LIN {X 0,Y 367.15,Z 1229.112,A -85,B 0,C 180,E1 18985.265,E2 18985.265} C_VEL
LIN {X 0,Y 367.339,Z 1230.535,A -85,B 0,C 180,E1 18990,E2 18990} C_VEL
LIN {X 0,Y 367.173,Z 1229.12,A -85,B 0,C 180,E1 18994.734,E2 18994.734} C_VEL
LIN {X 0,Y 367.735,Z 1223.43,A -85,B 0,C 180,E1 19000.686,E2 19000.686} C_VEL
LIN {X 0,Y 369.708,Z 1212.061,A -85,B 0,C 180,E1 19007.286,E2 19007.286} C_VEL
LIN {X 0,Y 374.711,Z 1193.004,A -85,B 0,C 180,E1 19014.404,E2 19014.404} C_VEL
LIN {X 0,Y 382.386,Z 1169.034,A -85,B 0,C 180,E1 19020.677,E2 19020.677} C_VEL
LIN {X 0,Y 392.699,Z 1139.664,A -85,B 0,C 180,E1 19026.255,E2 19026.255} C_VEL
LIN {X 0,Y 404.453,Z 1104.956,A -85,B 0,C 180,E1 19031.092,E2 19031.092} C_VEL
LIN {X 0,Y 416.185,Z 1066.688,A -85,B 0,C 180,E1 19034.968,E2 19034.968} C_VEL
LIN {X 0,Y 426.949,Z 1024.996,A -85,B 0,C 180,E1 19037.984,E2 19037.984} C_VEL
LIN {X 0,Y 432.113,Z 1000.704,A -85,B 0,C 180,E1 19039.291,E2 19039.291} C_VEL
LIN {X 0,Y 431.695,Z 993.378,A -85,B 0,C 180,E1 19039.909,E2 19039.909} C_VEL
LIN {X 0,Y 427.323,Z 982.88,A -85,B 0,C 180,E1 19041.274,E2 19041.274} C_VEL
LIN {X 0,Y 415.984,Z 952.064,A -85,B 0,C 180,E1 19044.997,E2 19044.997} C_VEL
LIN {X 0,Y 400.09,Z 921.403,A -85,B 0,C 180,E1 19049.492,E2 19049.492} C_VEL
LIN {X 0,Y 385.069,Z 898.25,A -85,B 0,C 180,E1 19053.963,E2 19053.963} C_VEL
LIN {X 0,Y 372.467,Z 880.115,A -85,B 0,C 180,E1 19058.525,E2 19058.525} C_VEL
LIN {X 0,Y 367.434,Z 873.394,A -85,B 0,C 180,E1 19060.66,E2 19060.66} C_VEL
LIN {X 0,Y 363.503,Z 867.579,A -85,B 0,C 180,E1 19062.545,E2 19062.545} C_VEL
LIN {X 0,Y 358.526,Z 862.168,A -85,B 0,C 180,E1 19065.154,E2 19065.154} C_VEL
LIN {X 0,Y 358.075,Z 859.31,A -85,B 0,C 180,E1 19065.699,E2 19065.699} C_VEL
LIN {X 0,Y 358.617,Z 859.31,A -85,B 0,C 180,E1 19072.716,E2 19072.716} C_VEL
LIN {X 0,Y 359.258,Z 859.31,A -85,B 0,C 180,E1 19079.997,E2 19079.997} C_VEL
LIN {X 0,Y 358.638,Z 859.31,A -85,B 0,C 180,E1 19087.277,E2 19087.277} C_VEL
LIN {X 0,Y 358.029,Z 859.31,A -85,B 0,C 180,E1 19094.703,E2 19094.703} C_VEL
LIN {X 0,Y 357.661,Z 859.332,A -85,B 0,C 180,E1 19100.287,E2 19100.287} C_VEL
LIN {X 0,Y 359.157,Z 864.008,A -85,B 0,C 180,E1 19101.329,E2 19101.329} C_VEL
LIN {X 0,Y 363.357,Z 867.747,A -85,B 0,C 180,E1 19103.444,E2 19103.444} C_VEL
LIN {X 0,Y 366.991,Z 873.322,A -85,B 0,C 180,E1 19105.191,E2 19105.191} C_VEL
LIN {X 0,Y 369.225,Z 876.271,A -85,B 0,C 180,E1 19106.168,E2 19106.168} C_VEL
LIN {X 0,Y 379.086,Z 889.509,A -85,B 0,C 180,E1 19109.965,E2 19109.965} C_VEL
LIN {X 0,Y 395.189,Z 912.841,A -85,B 0,C 180,E1 19115,E2 19115} C_VEL
LIN {X 0,Y 413.421,Z 943.358,A -85,B 0,C 180,E1 19119.705,E2 19119.705} C_VEL
LIN {X 0,Y 427.964,Z 974.626,A -85,B 0,C 180,E1 19123.471,E2 19123.471} C_VEL
LIN {X 0,Y 431.637,Z 986.503,A -85,B 0,C 180,E1 19124.663,E2 19124.663} C_VEL
LIN {X 0,Y 424.084,Z 1024.913,A -85,B 0,C 180,E1 19126.278,E2 19126.278} C_VEL
LIN {X 0,Y 414.384,Z 1061.767,A -85,B 0,C 180,E1 19128.631,E2 19128.631} C_VEL
LIN {X 0,Y 403.385,Z 1095.493,A -85,B 0,C 180,E1 19131.699,E2 19131.699} C_VEL
LIN {X 0,Y 391.865,Z 1125.986,A -85,B 0,C 180,E1 19135.561,E2 19135.561} C_VEL
LIN {X 0,Y 380.389,Z 1153.684,A -85,B 0,C 180,E1 19140.465,E2 19140.465} C_VEL
LIN {X 0,Y 371.321,Z 1175.527,A -85,B 0,C 180,E1 19145.916,E2 19145.916} C_VEL
LIN {X 0,Y 364.796,Z 1192.186,A -85,B 0,C 180,E1 19151.849,E2 19151.849} C_VEL
LIN {X 0,Y 361.198,Z 1203.353,A -85,B 0,C 180,E1 19157.892,E2 19157.892} C_VEL
LIN {X 0,Y 359.855,Z 1208.915,A -85,B 0,C 180,E1 19162.743,E2 19162.743} C_VEL
LIN {X 0,Y 359.413,Z 1211.64,A -85,B 0,C 180,E1 19167.584,E2 19167.584} C_VEL
LIN {X 0,Y 359.465,Z 1211.596,A -85,B 0,C 180,E1 19172.416,E2 19172.416} C_VEL
LIN {X 0,Y 360.028,Z 1208.022,A -85,B 0,C 180,E1 19178.09,E2 19178.09} C_VEL
LIN {X 0,Y 362.386,Z 1199.251,A -85,B 0,C 180,E1 19184.53,E2 19184.53} C_VEL
LIN {X 0,Y 367.067,Z 1185.895,A -85,B 0,C 180,E1 19190.542,E2 19190.542} C_VEL
LIN {X 0,Y 374.831,Z 1166.721,A -85,B 0,C 180,E1 19196.404,E2 19196.404} C_VEL
LIN {X 0,Y 385.163,Z 1142.05,A -85,B 0,C 180,E1 19201.695,E2 19201.695} C_VEL
LIN {X 0,Y 396.787,Z 1113.062,A -85,B 0,C 180,E1 19206.125,E2 19206.125} C_VEL
LIN {X 0,Y 408.628,Z 1079.698,A -85,B 0,C 180,E1 19209.768,E2 19209.768} C_VEL
LIN {X 0,Y 419.448,Z 1043.217,A -85,B 0,C 180,E1 19212.567,E2 19212.567} C_VEL
LIN {X 0,Y 428.235,Z 1005.04,A -85,B 0,C 180,E1 19214.553,E2 19214.553} C_VEL
LIN {X 0,Y 431.34,Z 984.283,A -85,B 0,C 180,E1 19215.383,E2 19215.383} C_VEL
LIN {X 0,Y 417.794,Z 951.743,A -85,B 0,C 180,E1 19219.089,E2 19219.089} C_VEL
LIN {X 0,Y 400.846,Z 921.844,A -85,B 0,C 180,E1 19223.316,E2 19223.316} C_VEL
LIN {X 0,Y 385.133,Z 898.179,A -85,B 0,C 180,E1 19227.847,E2 19227.847} C_VEL
LIN {X 0,Y 375.352,Z 884.709,A -85,B 0,C 180,E1 19231.201,E2 19231.201} C_VEL
LIN {X 0,Y 371.503,Z 879.558,A -85,B 0,C 180,E1 19232.697,E2 19232.697} C_VEL
LIN {X 0,Y 367.256,Z 873.532,A -85,B 0,C 180,E1 19234.502,E2 19234.502} C_VEL
LIN {X 0,Y 363.334,Z 867.894,A -85,B 0,C 180,E1 19236.349,E2 19236.349} C_VEL
LIN {X 0,Y 357.895,Z 861.738,A -85,B 0,C 180,E1 19239.2,E2 19239.2} C_VEL
LIN {X 0,Y 357.537,Z 859.31,A -85,B 0,C 180,E1 19239.568,E2 19239.568} C_VEL
LIN {X 0,Y 358.034,Z 859.31,A -85,B 0,C 180,E1 19246.761,E2 19246.761} C_VEL
LIN {X 0,Y 358.648,Z 859.31,A -85,B 0,C 180,E1 19252.723,E2 19252.723} C_VEL
LIN {X 0,Y 359.263,Z 859.31,A -85,B 0,C 180,E1 19260.003,E2 19260.003} C_VEL
LIN {X 0,Y 358.62,Z 859.31,A -85,B 0,C 180,E1 19267.284,E2 19267.284} C_VEL
LIN {X 0,Y 358.065,Z 859.874,A -85,B 0,C 180,E1 19274.607,E2 19274.607} C_VEL
LIN {X 0,Y 360.037,Z 864.711,A -85,B 0,C 180,E1 19275.876,E2 19275.876} C_VEL
LIN {X 0,Y 363.614,Z 867.802,A -85,B 0,C 180,E1 19277.621,E2 19277.621} C_VEL
LIN {X 0,Y 367.718,Z 873.561,A -85,B 0,C 180,E1 19279.559,E2 19279.559} C_VEL
LIN {X 0,Y 378.979,Z 889.438,A -85,B 0,C 180,E1 19284.034,E2 19284.034} C_VEL
LIN {X 0,Y 394.773,Z 912.854,A -85,B 0,C 180,E1 19289.06,E2 19289.06} C_VEL
LIN {X 0,Y 410.649,Z 941.029,A -85,B 0,C 180,E1 19293.521,E2 19293.521} C_VEL
LIN {X 0,Y 423.673,Z 972.018,A -85,B 0,C 180,E1 19297.488,E2 19297.488} C_VEL
LIN {X 0,Y 428.621,Z 990.013,A -85,B 0,C 180,E1 19299.444,E2 19299.444} C_VEL
LIN {X 0,Y 419.597,Z 1031.759,A -85,B 0,C 180,E1 19301.677,E2 19301.677} C_VEL
LIN {X 0,Y 409.092,Z 1070.519,A -85,B 0,C 180,E1 19304.638,E2 19304.638} C_VEL
LIN {X 0,Y 397.997,Z 1105.491,A -85,B 0,C 180,E1 19308.274,E2 19308.274} C_VEL
LIN {X 0,Y 386.322,Z 1138.586,A -85,B 0,C 180,E1 19312.91,E2 19312.91} C_VEL
LIN {X 0,Y 375.347,Z 1168.687,A -85,B 0,C 180,E1 19318.683,E2 19318.683} C_VEL
LIN {X 0,Y 367.176,Z 1193.104,A -85,B 0,C 180,E1 19325.193,E2 19325.193} C_VEL
LIN {X 0,Y 361.975,Z 1211.802,A -85,B 0,C 180,E1 19332.332,E2 19332.332} C_VEL
LIN {X 0,Y 359.893,Z 1223.198,A -85,B 0,C 180,E1 19339.078,E2 19339.078} C_VEL
LIN {X 0,Y 359.249,Z 1228.908,A -85,B 0,C 180,E1 19345.161,E2 19345.161} C_VEL
LIN {X 0,Y 359.439,Z 1230.334,A -85,B 0,C 180,E1 19350,E2 19350} C_VEL
LIN {X 0,Y 359.271,Z 1228.917,A -85,B 0,C 180,E1 19354.839,E2 19354.839} C_VEL
LIN {X 0,Y 359.87,Z 1223.22,A -85,B 0,C 180,E1 19360.922,E2 19360.922} C_VEL
LIN {X 0,Y 362,Z 1211.84,A -85,B 0,C 180,E1 19367.666,E2 19367.666} C_VEL
LIN {X 0,Y 367.136,Z 1193.199,A -85,B 0,C 180,E1 19374.793,E2 19374.793} C_VEL
LIN {X 0,Y 375.333,Z 1168.767,A -85,B 0,C 180,E1 19381.318,E2 19381.318} C_VEL
LIN {X 0,Y 386.374,Z 1138.707,A -85,B 0,C 180,E1 19387.083,E2 19387.083} C_VEL
LIN {X 0,Y 398.576,Z 1103.925,A -85,B 0,C 180,E1 19391.942,E2 19391.942} C_VEL
LIN {X 0,Y 410.79,Z 1065.255,A -85,B 0,C 180,E1 19395.85,E2 19395.85} C_VEL
LIN {X 0,Y 422.083,Z 1022.173,A -85,B 0,C 180,E1 19398.93,E2 19398.93} C_VEL
LIN {X 0,Y 428.825,Z 988.285,A -85,B 0,C 180,E1 19400.675,E2 19400.675} C_VEL
LIN {X 0,Y 427.323,Z 982.88,A -85,B 0,C 180,E1 19401.274,E2 19401.274} C_VEL
LIN {X 0,Y 422.821,Z 974.863,A -85,B 0,C 180,E1 19402.536,E2 19402.536} C_VEL
LIN {X 0,Y 414.499,Z 964.488,A -85,B 0,C 180,E1 19404.576,E2 19404.576} C_VEL
LIN {X 0,Y 413.821,Z 962.982,A -85,B 0,C 180,E1 19404.78,E2 19404.78} C_VEL
LIN {X 0,Y 399.432,Z 932.446,A -85,B 0,C 180,E1 19409.199,E2 19409.199} C_VEL
LIN {X 0,Y 383.451,Z 906.31,A -85,B 0,C 180,E1 19414.081,E2 19414.081} C_VEL
LIN {X 0,Y 369.915,Z 886.915,A -85,B 0,C 180,E1 19419.077,E2 19419.077} C_VEL
LIN {X 0,Y 364.832,Z 880.19,A -85,B 0,C 180,E1 19421.303,E2 19421.303} C_VEL
LIN {X 0,Y 360.151,Z 873.645,A -85,B 0,C 180,E1 19423.659,E2 19423.659} C_VEL
LIN {X 0,Y 356.32,Z 868.398,A -85,B 0,C 180,E1 19425.853,E2 19425.853} C_VEL
LIN {X 0,Y 355.113,Z 866.619,A -85,B 0,C 180,E1 19426.621,E2 19426.621} C_VEL
LIN {X 0,Y 350.857,Z 862.095,A -85,B 0,C 180,E1 19429.58,E2 19429.58} C_VEL
LIN {X 0,Y 350.463,Z 859.31,A -85,B 0,C 180,E1 19430.354,E2 19430.354} C_VEL
LIN {X 0,Y 351.103,Z 859.31,A -85,B 0,C 180,E1 19437.524,E2 19437.524} C_VEL
LIN {X 0,Y 351.143,Z 859.31,A -85,B 0,C 180,E1 19442.469,E2 19442.469} C_VEL
LIN {X 0,Y 350.438,Z 859.31,A -85,B 0,C 180,E1 19449.954,E2 19449.954} C_VEL
LIN {X 0,Y 350.018,Z 859.869,A -85,B 0,C 180,E1 19455.691,E2 19455.691} C_VEL
LIN {X 0,Y 352.008,Z 864.599,A -85,B 0,C 180,E1 19457.444,E2 19457.444} C_VEL
LIN {X 0,Y 355.863,Z 867.923,A -85,B 0,C 180,E1 19459.907,E2 19459.907} C_VEL
LIN {X 0,Y 359.622,Z 873.5,A -85,B 0,C 180,E1 19462.115,E2 19462.115} C_VEL
LIN {X 0,Y 361.689,Z 875.929,A -85,B 0,C 180,E1 19463.174,E2 19463.174} C_VEL
LIN {X 0,Y 367.943,Z 884.815,A -85,B 0,C 180,E1 19466.102,E2 19466.102} C_VEL
LIN {X 0,Y 377.036,Z 897.067,A -85,B 0,C 180,E1 19469.647,E2 19469.647} C_VEL
LIN {X 0,Y 392.135,Z 919.205,A -85,B 0,C 180,E1 19474.485,E2 19474.485} C_VEL
LIN {X 0,Y 409.719,Z 949.301,A -85,B 0,C 180,E1 19479.203,E2 19479.203} C_VEL
LIN {X 0,Y 423.434,Z 980.427,A -85,B 0,C 180,E1 19483.058,E2 19483.058} C_VEL
LIN {X 0,Y 425.993,Z 988.977,A -85,B 0,C 180,E1 19483.955,E2 19483.955} C_VEL
LIN {X 0,Y 418.022,Z 1027.436,A -85,B 0,C 180,E1 19485.628,E2 19485.628} C_VEL
LIN {X 0,Y 407.954,Z 1064.073,A -85,B 0,C 180,E1 19488.042,E2 19488.042} C_VEL
LIN {X 0,Y 396.34,Z 1098.126,A -85,B 0,C 180,E1 19491.241,E2 19491.241} C_VEL
LIN {X 0,Y 384.591,Z 1128,A -85,B 0,C 180,E1 19495.159,E2 19495.159} C_VEL
LIN {X 0,Y 373.441,Z 1153.942,A -85,B 0,C 180,E1 19499.859,E2 19499.859} C_VEL
LIN {X 0,Y 364.005,Z 1175.757,A -85,B 0,C 180,E1 19505.4,E2 19505.4} C_VEL
LIN {X 0,Y 357.194,Z 1192.404,A -85,B 0,C 180,E1 19511.448,E2 19511.448} C_VEL
LIN {X 0,Y 353.418,Z 1203.561,A -85,B 0,C 180,E1 19517.621,E2 19517.621} C_VEL
LIN {X 0,Y 351.979,Z 1209.12,A -85,B 0,C 180,E1 19522.58,E2 19522.58} C_VEL
LIN {X 0,Y 351.514,Z 1211.843,A -85,B 0,C 180,E1 19527.53,E2 19527.53} C_VEL
LIN {X 0,Y 351.564,Z 1211.798,A -85,B 0,C 180,E1 19532.471,E2 19532.471} C_VEL
LIN {X 0,Y 352.232,Z 1208.057,A -85,B 0,C 180,E1 19538.455,E2 19538.455} C_VEL
LIN {X 0,Y 354.68,Z 1199.462,A -85,B 0,C 180,E1 19544.853,E2 19544.853} C_VEL
LIN {X 0,Y 359.6,Z 1186.123,A -85,B 0,C 180,E1 19550.988,E2 19550.988} C_VEL
LIN {X 0,Y 367.684,Z 1166.975,A -85,B 0,C 180,E1 19556.958,E2 19556.958} C_VEL
LIN {X 0,Y 378.689,Z 1141.618,A -85,B 0,C 180,E1 19562.46,E2 19562.46} C_VEL
LIN {X 0,Y 390.707,Z 1112.592,A -85,B 0,C 180,E1 19566.918,E2 19566.918} C_VEL
LIN {X 0,Y 402.592,Z 1080.169,A -85,B 0,C 180,E1 19570.486,E2 19570.486} C_VEL
LIN {X 0,Y 413.994,Z 1042.731,A -85,B 0,C 180,E1 19573.375,E2 19573.375} C_VEL
LIN {X 0,Y 423.128,Z 1003.727,A -85,B 0,C 180,E1 19575.393,E2 19575.393} C_VEL
LIN {X 0,Y 425.615,Z 987.109,A -85,B 0,C 180,E1 19576.086,E2 19576.086} C_VEL
LIN {X 0,Y 412.44,Z 954.819,A -85,B 0,C 180,E1 19579.919,E2 19579.919} C_VEL
LIN {X 0,Y 396.061,Z 925.668,A -85,B 0,C 180,E1 19584.252,E2 19584.252} C_VEL
LIN {X 0,Y 379.708,Z 900.578,A -85,B 0,C 180,E1 19589.262,E2 19589.262} C_VEL
LIN {X 0,Y 368.895,Z 886.075,A -85,B 0,C 180,E1 19593.314,E2 19593.314} C_VEL
LIN {X 0,Y 364.408,Z 880.099,A -85,B 0,C 180,E1 19595.276,E2 19595.276} C_VEL
LIN {X 0,Y 360.295,Z 873.963,A -85,B 0,C 180,E1 19597.34,E2 19597.34} C_VEL
LIN {X 0,Y 355.922,Z 868.494,A -85,B 0,C 180,E1 19599.772,E2 19599.772} C_VEL
LIN {X 0,Y 354.505,Z 866.563,A -85,B 0,C 180,E1 19600.663,E2 19600.663} C_VEL
LIN {X 0,Y 350.327,Z 861.978,A -85,B 0,C 180,E1 19603.599,E2 19603.599} C_VEL
LIN {X 0,Y 349.914,Z 859.31,A -85,B 0,C 180,E1 19604.305,E2 19604.305} C_VEL
LIN {X 0,Y 350.437,Z 859.31,A -85,B 0,C 180,E1 19610.046,E2 19610.046} C_VEL
LIN {X 0,Y 351.109,Z 859.31,A -85,B 0,C 180,E1 19617.531,E2 19617.531} C_VEL
LIN {X 0,Y 351.148,Z 859.31,A -85,B 0,C 180,E1 19622.476,E2 19622.476} C_VEL
LIN {X 0,Y 350.42,Z 859.698,A -85,B 0,C 180,E1 19630.118,E2 19630.118} C_VEL
LIN {X 0,Y 352.122,Z 864.387,A -85,B 0,C 180,E1 19631.638,E2 19631.638} C_VEL
LIN {X 0,Y 356.14,Z 867.806,A -85,B 0,C 180,E1 19634.158,E2 19634.158} C_VEL
LIN {X 0,Y 359.617,Z 873.291,A -85,B 0,C 180,E1 19636.209,E2 19636.209} C_VEL
LIN {X 0,Y 361.893,Z 875.863,A -85,B 0,C 180,E1 19637.356,E2 19637.356} C_VEL
LIN {X 0,Y 367.733,Z 884.15,A -85,B 0,C 180,E1 19640.107,E2 19640.107} C_VEL
LIN {X 0,Y 376.638,Z 896.626,A -85,B 0,C 180,E1 19643.641,E2 19643.641} C_VEL
LIN {X 0,Y 391.562,Z 919.088,A -85,B 0,C 180,E1 19648.53,E2 19648.53} C_VEL
LIN {X 0,Y 406.621,Z 946.779,A -85,B 0,C 180,E1 19653.019,E2 19653.019} C_VEL
LIN {X 0,Y 418.988,Z 977.742,A -85,B 0,C 180,E1 19657.083,E2 19657.083} C_VEL
LIN {X 0,Y 422.934,Z 992.326,A -85,B 0,C 180,E1 19658.745,E2 19658.745} C_VEL
LIN {X 0,Y 412.869,Z 1036.702,A -85,B 0,C 180,E1 19661.203,E2 19661.203} C_VEL
LIN {X 0,Y 400.633,Z 1079.007,A -85,B 0,C 180,E1 19664.64,E2 19664.64} C_VEL
LIN {X 0,Y 387.942,Z 1116.268,A -85,B 0,C 180,E1 19668.892,E2 19668.892} C_VEL
LIN {X 0,Y 375.255,Z 1150.031,A -85,B 0,C 180,E1 19674.225,E2 19674.225} C_VEL
LIN {X 0,Y 365.282,Z 1177.147,A -85,B 0,C 180,E1 19680.145,E2 19680.145} C_VEL
LIN {X 0,Y 357.663,Z 1199.514,A -85,B 0,C 180,E1 19686.927,E2 19686.927} C_VEL
LIN {X 0,Y 353.375,Z 1215.207,A -85,B 0,C 180,E1 19693.816,E2 19693.816} C_VEL
LIN {X 0,Y 351.812,Z 1224.499,A -85,B 0,C 180,E1 19700.079,E2 19700.079} C_VEL
LIN {X 0,Y 351.35,Z 1228.705,A -85,B 0,C 180,E1 19705.051,E2 19705.051} C_VEL
LIN {X 0,Y 351.54,Z 1230.132,A -85,B 0,C 180,E1 19710,E2 19710} C_VEL
LIN {X 0,Y 351.37,Z 1228.714,A -85,B 0,C 180,E1 19714.948,E2 19714.948} C_VEL
LIN {X 0,Y 352.005,Z 1223.01,A -85,B 0,C 180,E1 19721.169,E2 19721.169} C_VEL
LIN {X 0,Y 354.296,Z 1211.619,A -85,B 0,C 180,E1 19728.064,E2 19728.064} C_VEL
LIN {X 0,Y 359.767,Z 1192.96,A -85,B 0,C 180,E1 19735.337,E2 19735.337} C_VEL
LIN {X 0,Y 368.369,Z 1168.5,A -85,B 0,C 180,E1 19741.979,E2 19741.979} C_VEL
LIN {X 0,Y 379.889,Z 1138.391,A -85,B 0,C 180,E1 19747.826,E2 19747.826} C_VEL
LIN {X 0,Y 392.422,Z 1103.855,A -85,B 0,C 180,E1 19752.701,E2 19752.701} C_VEL
LIN {X 0,Y 405.166,Z 1064.689,A -85,B 0,C 180,E1 19756.68,E2 19756.68} C_VEL
LIN {X 0,Y 416.483,Z 1022.91,A -85,B 0,C 180,E1 19759.679,E2 19759.679} C_VEL
LIN {X 0,Y 423.112,Z 991.352,A -85,B 0,C 180,E1 19761.329,E2 19761.329} C_VEL
LIN {X 0,Y 413.821,Z 962.982,A -85,B 0,C 180,E1 19764.78,E2 19764.78} C_VEL
LIN {X 0,Y 408.724,Z 955.768,A -85,B 0,C 180,E1 19766.131,E2 19766.131} C_VEL
LIN {X 0,Y 399.285,Z 945.576,A -85,B 0,C 180,E1 19768.576,E2 19768.576} C_VEL
LIN {X 0,Y 384.747,Z 919.229,A -85,B 0,C 180,E1 19773.231,E2 19773.231} C_VEL
LIN {X 0,Y 368.413,Z 894.706,A -85,B 0,C 180,E1 19779.224,E2 19779.224} C_VEL
LIN {X 0,Y 358.317,Z 881.083,A -85,B 0,C 180,E1 19784.046,E2 19784.046} C_VEL
LIN {X 0,Y 354.379,Z 875.295,A -85,B 0,C 180,E1 19786.398,E2 19786.398} C_VEL
LIN {X 0,Y 349.218,Z 869.207,A -85,B 0,C 180,E1 19790.083,E2 19790.083} C_VEL
LIN {X 0,Y 348.367,Z 866.925,A -85,B 0,C 180,E1 19790.927,E2 19790.927} C_VEL
LIN {X 0,Y 343.482,Z 861.831,A -85,B 0,C 180,E1 19796.52,E2 19796.52} C_VEL
LIN {X 0,Y 343.23,Z 859.31,A -85,B 0,C 180,E1 19797.783,E2 19797.783} C_VEL
LIN {X 0,Y 343.227,Z 859.31,A -85,B 0,C 180,E1 19802.526,E2 19802.526} C_VEL
LIN {X 0,Y 342.745,Z 859.975,A -85,B 0,C 180,E1 19807.856,E2 19807.856} C_VEL
LIN {X 0,Y 345.119,Z 865.303,A -85,B 0,C 180,E1 19812.031,E2 19812.031} C_VEL
LIN {X 0,Y 348.552,Z 867.994,A -85,B 0,C 180,E1 19815.346,E2 19815.346} C_VEL
LIN {X 0,Y 352.066,Z 873.596,A -85,B 0,C 180,E1 19818.174,E2 19818.174} C_VEL
LIN {X 0,Y 354.361,Z 875.948,A -85,B 0,C 180,E1 19819.639,E2 19819.639} C_VEL
LIN {X 0,Y 359.026,Z 881.65,A -85,B 0,C 180,E1 19822.315,E2 19822.315} C_VEL
LIN {X 0,Y 373.94,Z 902.767,A -85,B 0,C 180,E1 19828.918,E2 19828.918} C_VEL
LIN {X 0,Y 389.418,Z 926.115,A -85,B 0,C 180,E1 19834.056,E2 19834.056} C_VEL
LIN {X 0,Y 405.851,Z 955.267,A -85,B 0,C 180,E1 19838.721,E2 19838.721} C_VEL
LIN {X 0,Y 418.768,Z 986.191,A -85,B 0,C 180,E1 19842.651,E2 19842.651} C_VEL
LIN {X 0,Y 420.308,Z 992.169,A -85,B 0,C 180,E1 19843.256,E2 19843.256} C_VEL
LIN {X 0,Y 411.574,Z 1031.755,A -85,B 0,C 180,E1 19845.055,E2 19845.055} C_VEL
LIN {X 0,Y 400.039,Z 1070.982,A -85,B 0,C 180,E1 19847.802,E2 19847.802} C_VEL
LIN {X 0,Y 387.602,Z 1105.211,A -85,B 0,C 180,E1 19851.281,E2 19851.281} C_VEL
LIN {X 0,Y 374.579,Z 1136.428,A -85,B 0,C 180,E1 19855.8,E2 19855.8} C_VEL
LIN {X 0,Y 362.821,Z 1162.416,A -85,B 0,C 180,E1 19861.134,E2 19861.134} C_VEL
LIN {X 0,Y 354.356,Z 1181.426,A -85,B 0,C 180,E1 19866.629,E2 19866.629} C_VEL
LIN {X 0,Y 347.87,Z 1197.306,A -85,B 0,C 180,E1 19873.333,E2 19873.333} C_VEL
LIN {X 0,Y 344.701,Z 1206.912,A -85,B 0,C 180,E1 19879.873,E2 19879.873} C_VEL
LIN {X 0,Y 343.776,Z 1211.03,A -85,B 0,C 180,E1 19884.943,E2 19884.943} C_VEL
LIN {X 0,Y 343.666,Z 1212.365,A -85,B 0,C 180,E1 19890,E2 19890} C_VEL
LIN {X 0,Y 343.792,Z 1210.956,A -85,B 0,C 180,E1 19895.058,E2 19895.058} C_VEL
LIN {X 0,Y 345.209,Z 1205.29,A -85,B 0,C 180,E1 19901.393,E2 19901.393} C_VEL
LIN {X 0,Y 349.176,Z 1193.679,A -85,B 0,C 180,E1 19908.338,E2 19908.338} C_VEL
LIN {X 0,Y 356.801,Z 1175.663,A -85,B 0,C 180,E1 19915.131,E2 19915.131} C_VEL
LIN {X 0,Y 367.379,Z 1152.445,A -85,B 0,C 180,E1 19921.036,E2 19921.036} C_VEL
LIN {X 0,Y 379.761,Z 1124.211,A -85,B 0,C 180,E1 19926.054,E2 19926.054} C_VEL
LIN {X 0,Y 392.566,Z 1091.951,A -85,B 0,C 180,E1 19930.101,E2 19930.101} C_VEL
LIN {X 0,Y 404.763,Z 1055.846,A -85,B 0,C 180,E1 19933.27,E2 19933.27} C_VEL
LIN {X 0,Y 414.816,Z 1018.042,A -85,B 0,C 180,E1 19935.553,E2 19935.553} C_VEL
LIN {X 0,Y 419.92,Z 989.876,A -85,B 0,C 180,E1 19936.816,E2 19936.816} C_VEL
LIN {X 0,Y 407.158,Z 958.008,A -85,B 0,C 180,E1 19940.768,E2 19940.768} C_VEL
LIN {X 0,Y 391.258,Z 929.144,A -85,B 0,C 180,E1 19945.251,E2 19945.251} C_VEL
LIN {X 0,Y 375.727,Z 905.574,A -85,B 0,C 180,E1 19950.24,E2 19950.24} C_VEL
LIN {X 0,Y 363.526,Z 888.276,A -85,B 0,C 180,E1 19955.212,E2 19955.212} C_VEL
LIN {X 0,Y 357.749,Z 880.867,A -85,B 0,C 180,E1 19958.108,E2 19958.108} C_VEL
LIN {X 0,Y 352.815,Z 874.13,A -85,B 0,C 180,E1 19961.088,E2 19961.088} C_VEL
LIN {X 0,Y 348.623,Z 868.766,A -85,B 0,C 180,E1 19964.206,E2 19964.206} C_VEL
LIN {X 0,Y 347.596,Z 866.844,A -85,B 0,C 180,E1 19965.156,E2 19965.156} C_VEL
LIN {X 0,Y 342.899,Z 861.607,A -85,B 0,C 180,E1 19970.708,E2 19970.708} C_VEL
LIN {X 0,Y 342.649,Z 859.31,A -85,B 0,C 180,E1 19971.742,E2 19971.742} C_VEL
LIN {X 0,Y 343.194,Z 859.31,A -85,B 0,C 180,E1 19977.474,E2 19977.474} C_VEL
LIN {X 0,Y 343.175,Z 860.095,A -85,B 0,C 180,E1 19983.246,E2 19983.246} C_VEL
LIN {X 0,Y 345.821,Z 865.525,A -85,B 0,C 180,E1 19987.04,E2 19987.04} C_VEL
LIN {X 0,Y 348.86,Z 868.02,A -85,B 0,C 180,E1 19989.769,E2 19989.769} C_VEL
LIN {X 0,Y 352.254,Z 873.421,A -85,B 0,C 180,E1 19992.421,E2 19992.421} C_VEL
LIN {X 0,Y 354.487,Z 875.664,A -85,B 0,C 180,E1 19993.834,E2 19993.834} C_VEL
LIN {X 0,Y 358.94,Z 881.458,A -85,B 0,C 180,E1 19996.398,E2 19996.398} C_VEL
LIN {X 0,Y 369.672,Z 896.846,A -85,B 0,C 180,E1 20001.409,E2 20001.409} C_VEL
LIN {X 0,Y 384.948,Z 919.742,A -85,B 0,C 180,E1 20006.912,E2 20006.912} C_VEL
LIN {X 0,Y 399.196,Z 945.574,A -85,B 0,C 180,E1 20011.456,E2 20011.456} C_VEL
LIN {X 0,Y 411.296,Z 974.691,A -85,B 0,C 180,E1 20015.577,E2 20015.577} C_VEL
LIN {X 0,Y 417.119,Z 995.397,A -85,B 0,C 180,E1 20018.069,E2 20018.069} C_VEL
LIN {X 0,Y 406.939,Z 1038.429,A -85,B 0,C 180,E1 20020.509,E2 20020.509} C_VEL
LIN {X 0,Y 394.695,Z 1079.379,A -85,B 0,C 180,E1 20023.886,E2 20023.886} C_VEL
LIN {X 0,Y 382.128,Z 1115.152,A -85,B 0,C 180,E1 20027.99,E2 20027.99} C_VEL
LIN {X 0,Y 369.263,Z 1148.207,A -85,B 0,C 180,E1 20033.195,E2 20033.195} C_VEL
LIN {X 0,Y 358.197,Z 1176.882,A -85,B 0,C 180,E1 20039.493,E2 20039.493} C_VEL
LIN {X 0,Y 350.13,Z 1199.472,A -85,B 0,C 180,E1 20046.476,E2 20046.476} C_VEL
LIN {X 0,Y 345.378,Z 1216.191,A -85,B 0,C 180,E1 20054.085,E2 20054.085} C_VEL
LIN {X 0,Y 343.798,Z 1225.573,A -85,B 0,C 180,E1 20061.126,E2 20061.126} C_VEL
LIN {X 0,Y 343.566,Z 1229.569,A -85,B 0,C 180,E1 20067.472,E2 20067.472} C_VEL
LIN {X 0,Y 343.558,Z 1229.571,A -85,B 0,C 180,E1 20072.528,E2 20072.528} C_VEL
LIN {X 0,Y 343.784,Z 1225.593,A -85,B 0,C 180,E1 20078.874,E2 20078.874} C_VEL
LIN {X 0,Y 345.428,Z 1216.227,A -85,B 0,C 180,E1 20085.912,E2 20085.912} C_VEL
LIN {X 0,Y 350.103,Z 1199.529,A -85,B 0,C 180,E1 20093.525,E2 20093.525} C_VEL
LIN {X 0,Y 358.191,Z 1176.962,A -85,B 0,C 180,E1 20100.507,E2 20100.507} C_VEL
LIN {X 0,Y 369.279,Z 1148.306,A -85,B 0,C 180,E1 20106.808,E2 20106.808} C_VEL
LIN {X 0,Y 382.144,Z 1115.276,A -85,B 0,C 180,E1 20112.015,E2 20112.015} C_VEL
LIN {X 0,Y 395.398,Z 1077.37,A -85,B 0,C 180,E1 20116.333,E2 20116.333} C_VEL
LIN {X 0,Y 407.775,Z 1035.881,A -85,B 0,C 180,E1 20119.67,E2 20119.67} C_VEL
LIN {X 0,Y 417.351,Z 994.067,A -85,B 0,C 180,E1 20122.039,E2 20122.039} C_VEL
LIN {X 0,Y 407.347,Z 963.466,A -85,B 0,C 180,E1 20125.936,E2 20125.936} C_VEL
LIN {X 0,Y 399.285,Z 945.576,A -85,B 0,C 180,E1 20128.576,E2 20128.576} C_VEL
LIN {X 0,Y 395.886,Z 941.099,A -85,B 0,C 180,E1 20129.545,E2 20129.545} C_VEL
LIN {X 0,Y 385.453,Z 931.977,A -85,B 0,C 180,E1 20132.478,E2 20132.478} C_VEL
LIN {X 0,Y 384.704,Z 930.725,A -85,B 0,C 180,E1 20132.724,E2 20132.724} C_VEL
LIN {X 0,Y 369.828,Z 907.382,A -85,B 0,C 180,E1 20138.127,E2 20138.127} C_VEL
LIN {X 0,Y 360.709,Z 894.477,A -85,B 0,C 180,E1 20142.191,E2 20142.191} C_VEL
LIN {X 0,Y 356.09,Z 888.129,A -85,B 0,C 180,E1 20144.656,E2 20144.656} C_VEL
LIN {X 0,Y 351.522,Z 881.565,A -85,B 0,C 180,E1 20147.553,E2 20147.553} C_VEL
LIN {X 0,Y 347.536,Z 876.057,A -85,B 0,C 180,E1 20150.668,E2 20150.668} C_VEL
LIN {X 0,Y 346.293,Z 874.345,A -85,B 0,C 180,E1 20151.823,E2 20151.823} C_VEL
LIN {X 0,Y 342.162,Z 868.741,A -85,B 0,C 180,E1 20157.221,E2 20157.221} C_VEL
LIN {X 0,Y 341.876,Z 867.092,A -85,B 0,C 180,E1 20158.092,E2 20158.092} C_VEL
LIN {X 0,Y 341.658,Z 867.792,A -85,B 0,C 180,E1 20167.564,E2 20167.564} C_VEL
LIN {X 0,Y 344.745,Z 873.663,A -85,B 0,C 180,E1 20172.689,E2 20172.689} C_VEL
LIN {X 0,Y 347.157,Z 875.681,A -85,B 0,C 180,E1 20175.003,E2 20175.003} C_VEL
LIN {X 0,Y 351.299,Z 881.641,A -85,B 0,C 180,E1 20178.311,E2 20178.311} C_VEL
LIN {X 0,Y 353.443,Z 884.854,A -85,B 0,C 180,E1 20179.743,E2 20179.743} C_VEL
LIN {X 0,Y 358.422,Z 891.44,A -85,B 0,C 180,E1 20182.6,E2 20182.6} C_VEL
LIN {X 0,Y 368.259,Z 905.192,A -85,B 0,C 180,E1 20187.149,E2 20187.149} C_VEL
LIN {X 0,Y 382.456,Z 926.004,A -85,B 0,C 180,E1 20192.274,E2 20192.274} C_VEL
LIN {X 0,Y 398.995,Z 955.04,A -85,B 0,C 180,E1 20197.327,E2 20197.327} C_VEL
LIN {X 0,Y 412.058,Z 985.78,A -85,B 0,C 180,E1 20201.5,E2 20201.5} C_VEL
LIN {X 0,Y 414.496,Z 995.633,A -85,B 0,C 180,E1 20202.559,E2 20202.559} C_VEL
LIN {X 0,Y 405.381,Z 1034.858,A -85,B 0,C 180,E1 20204.415,E2 20204.415} C_VEL
LIN {X 0,Y 394.096,Z 1071.77,A -85,B 0,C 180,E1 20207.06,E2 20207.06} C_VEL
LIN {X 0,Y 381.468,Z 1105.557,A -85,B 0,C 180,E1 20210.539,E2 20210.539} C_VEL
LIN {X 0,Y 368.628,Z 1135.395,A -85,B 0,C 180,E1 20214.867,E2 20214.867} C_VEL
LIN {X 0,Y 356.583,Z 1161.119,A -85,B 0,C 180,E1 20220.118,E2 20220.118} C_VEL
LIN {X 0,Y 346.843,Z 1182.013,A -85,B 0,C 180,E1 20226.234,E2 20226.234} C_VEL
LIN {X 0,Y 340.222,Z 1197.517,A -85,B 0,C 180,E1 20232.947,E2 20232.947} C_VEL
LIN {X 0,Y 336.879,Z 1207.118,A -85,B 0,C 180,E1 20239.635,E2 20239.635} C_VEL
LIN {X 0,Y 335.882,Z 1211.234,A -85,B 0,C 180,E1 20244.824,E2 20244.824} C_VEL
LIN {X 0,Y 335.767,Z 1212.567,A -85,B 0,C 180,E1 20250,E2 20250} C_VEL
LIN {X 0,Y 335.9,Z 1211.16,A -85,B 0,C 180,E1 20255.177,E2 20255.177} C_VEL
LIN {X 0,Y 337.405,Z 1205.496,A -85,B 0,C 180,E1 20261.66,E2 20261.66} C_VEL
LIN {X 0,Y 341.583,Z 1193.896,A -85,B 0,C 180,E1 20268.761,E2 20268.761} C_VEL
LIN {X 0,Y 349.556,Z 1175.893,A -85,B 0,C 180,E1 20275.69,E2 20275.69} C_VEL
LIN {X 0,Y 360.526,Z 1152.712,A -85,B 0,C 180,E1 20281.694,E2 20281.694} C_VEL
LIN {X 0,Y 373.346,Z 1124.544,A -85,B 0,C 180,E1 20286.774,E2 20286.774} C_VEL
LIN {X 0,Y 386.536,Z 1092.376,A -85,B 0,C 180,E1 20290.858,E2 20290.858} C_VEL
LIN {X 0,Y 398.952,Z 1056.855,A -85,B 0,C 180,E1 20294.013,E2 20294.013} C_VEL
LIN {X 0,Y 409.453,Z 1018.495,A -85,B 0,C 180,E1 20296.359,E2 20296.359} C_VEL
LIN {X 0,Y 414.42,Z 993.295,A -85,B 0,C 180,E1 20297.492,E2 20297.492} C_VEL
LIN {X 0,Y 402.582,Z 962.63,A -85,B 0,C 180,E1 20301.451,E2 20301.451} C_VEL
LIN {X 0,Y 387.595,Z 934.527,A -85,B 0,C 180,E1 20305.953,E2 20305.953} C_VEL
LIN {X 0,Y 372.426,Z 911.105,A -85,B 0,C 180,E1 20311.037,E2 20311.037} C_VEL
LIN {X 0,Y 360.913,Z 894.93,A -85,B 0,C 180,E1 20315.929,E2 20315.929} C_VEL
LIN {X 0,Y 355.904,Z 888.152,A -85,B 0,C 180,E1 20318.547,E2 20318.547} C_VEL
LIN {X 0,Y 351.234,Z 881.677,A -85,B 0,C 180,E1 20321.465,E2 20321.465} C_VEL
LIN {X 0,Y 347.03,Z 875.776,A -85,B 0,C 180,E1 20324.743,E2 20324.743} C_VEL
LIN {X 0,Y 341.598,Z 868.426,A -85,B 0,C 180,E1 20331.476,E2 20331.476} C_VEL
LIN {X 0,Y 341.277,Z 867.066,A -85,B 0,C 180,E1 20332.437,E2 20332.437} C_VEL
LIN {X 0,Y 341.947,Z 867.494,A -85,B 0,C 180,E1 20342.781,E2 20342.781} C_VEL
LIN {X 0,Y 344.73,Z 873.331,A -85,B 0,C 180,E1 20346.944,E2 20346.944} C_VEL
LIN {X 0,Y 347.398,Z 875.658,A -85,B 0,C 180,E1 20349.415,E2 20349.415} C_VEL
LIN {X 0,Y 351.274,Z 881.398,A -85,B 0,C 180,E1 20352.456,E2 20352.456} C_VEL
LIN {X 0,Y 353.287,Z 884.306,A -85,B 0,C 180,E1 20353.803,E2 20353.803} C_VEL
LIN {X 0,Y 358.673,Z 891.598,A -85,B 0,C 180,E1 20356.884,E2 20356.884} C_VEL
LIN {X 0,Y 367.62,Z 904.242,A -85,B 0,C 180,E1 20361.06,E2 20361.06} C_VEL
LIN {X 0,Y 381.953,Z 926.32,A -85,B 0,C 180,E1 20366.424,E2 20366.424} C_VEL
LIN {X 0,Y 395.623,Z 952.156,A -85,B 0,C 180,E1 20371.065,E2 20371.065} C_VEL
LIN {X 0,Y 406.919,Z 981.13,A -85,B 0,C 180,E1 20375.245,E2 20375.245} C_VEL
LIN {X 0,Y 411.345,Z 998.216,A -85,B 0,C 180,E1 20377.362,E2 20377.362} C_VEL
LIN {X 0,Y 401.36,Z 1039.063,A -85,B 0,C 180,E1 20379.719,E2 20379.719} C_VEL
LIN {X 0,Y 388.82,Z 1079.685,A -85,B 0,C 180,E1 20383.098,E2 20383.098} C_VEL
LIN {X 0,Y 375.298,Z 1116.87,A -85,B 0,C 180,E1 20387.445,E2 20387.445} C_VEL
LIN {X 0,Y 361.93,Z 1149.843,A -85,B 0,C 180,E1 20392.789,E2 20392.789} C_VEL
LIN {X 0,Y 351.16,Z 1176.617,A -85,B 0,C 180,E1 20398.814,E2 20398.814} C_VEL
LIN {X 0,Y 342.621,Z 1199.351,A -85,B 0,C 180,E1 20405.974,E2 20405.974} C_VEL
LIN {X 0,Y 337.619,Z 1215.971,A -85,B 0,C 180,E1 20413.709,E2 20413.709} C_VEL
LIN {X 0,Y 335.939,Z 1225.366,A -85,B 0,C 180,E1 20420.916,E2 20420.916} C_VEL
LIN {X 0,Y 335.655,Z 1229.366,A -85,B 0,C 180,E1 20427.412,E2 20427.412} C_VEL
LIN {X 0,Y 335.649,Z 1229.369,A -85,B 0,C 180,E1 20432.587,E2 20432.587} C_VEL
LIN {X 0,Y 335.901,Z 1225.386,A -85,B 0,C 180,E1 20439.084,E2 20439.084} C_VEL
LIN {X 0,Y 337.662,Z 1216.01,A -85,B 0,C 180,E1 20446.288,E2 20446.288} C_VEL
LIN {X 0,Y 342.602,Z 1199.418,A -85,B 0,C 180,E1 20454.023,E2 20454.023} C_VEL
LIN {X 0,Y 351.156,Z 1176.702,A -85,B 0,C 180,E1 20461.186,E2 20461.186} C_VEL
LIN {X 0,Y 362.39,Z 1148.935,A -85,B 0,C 180,E1 20467.41,E2 20467.41} C_VEL
LIN {X 0,Y 376.098,Z 1114.987,A -85,B 0,C 180,E1 20472.835,E2 20472.835} C_VEL
LIN {X 0,Y 389.464,Z 1077.991,A -85,B 0,C 180,E1 20477.096,E2 20477.096} C_VEL
LIN {X 0,Y 402.029,Z 1037.402,A -85,B 0,C 180,E1 20480.402,E2 20480.402} C_VEL
LIN {X 0,Y 411.526,Z 996.64,A -85,B 0,C 180,E1 20482.779,E2 20482.779} C_VEL
LIN {X 0,Y 401.943,Z 966.555,A -85,B 0,C 180,E1 20486.768,E2 20486.768} C_VEL
LIN {X 0,Y 388.795,Z 938.243,A -85,B 0,C 180,E1 20491.328,E2 20491.328} C_VEL
LIN {X 0,Y 384.704,Z 930.725,A -85,B 0,C 180,E1 20492.724,E2 20492.724} C_VEL
LIN {X 0,Y 379.562,Z 925.477,A -85,B 0,C 180,E1 20494.347,E2 20494.347} C_VEL
LIN {X 0,Y 370.671,Z 919.269,A -85,B 0,C 180,E1 20497.3,E2 20497.3} C_VEL
LIN {X 0,Y 359.567,Z 902.555,A -85,B 0,C 180,E1 20502.211,E2 20502.211} C_VEL
LIN {X 0,Y 353.913,Z 895.093,A -85,B 0,C 180,E1 20505.273,E2 20505.273} C_VEL
LIN {X 0,Y 349.863,Z 889.013,A -85,B 0,C 180,E1 20507.969,E2 20507.969} C_VEL
LIN {X 0,Y 345.959,Z 883.14,A -85,B 0,C 180,E1 20511.181,E2 20511.181} C_VEL
LIN {X 0,Y 340.957,Z 875.937,A -85,B 0,C 180,E1 20517.743,E2 20517.743} C_VEL
LIN {X 0,Y 340.133,Z 874.678,A -85,B 0,C 180,E1 20519.997,E2 20519.997} C_VEL
LIN {X 0,Y 340.609,Z 875.822,A -85,B 0,C 180,E1 20527.435,E2 20527.435} C_VEL
LIN {X 0,Y 344.167,Z 881.787,A -85,B 0,C 180,E1 20533.088,E2 20533.088} C_VEL
LIN {X 0,Y 345.937,Z 883.772,A -85,B 0,C 180,E1 20534.827,E2 20534.827} C_VEL
LIN {X 0,Y 351.502,Z 891.608,A -85,B 0,C 180,E1 20539.142,E2 20539.142} C_VEL
LIN {X 0,Y 357.059,Z 899.523,A -85,B 0,C 180,E1 20542.444,E2 20542.444} C_VEL
LIN {X 0,Y 366.157,Z 912.37,A -85,B 0,C 180,E1 20546.735,E2 20546.735} C_VEL
LIN {X 0,Y 379.978,Z 933.123,A -85,B 0,C 180,E1 20551.862,E2 20551.862} C_VEL
LIN {X 0,Y 395.057,Z 960.666,A -85,B 0,C 180,E1 20556.761,E2 20556.761} C_VEL
LIN {X 0,Y 407.079,Z 990.343,A -85,B 0,C 180,E1 20560.917,E2 20560.917} C_VEL
LIN {X 0,Y 408.992,Z 997.797,A -85,B 0,C 180,E1 20561.791,E2 20561.791} C_VEL
LIN {X 0,Y 400.046,Z 1035.031,A -85,B 0,C 180,E1 20563.58,E2 20563.58} C_VEL
LIN {X 0,Y 388.214,Z 1072.586,A -85,B 0,C 180,E1 20566.298,E2 20566.298} C_VEL
LIN {X 0,Y 374.888,Z 1107.033,A -85,B 0,C 180,E1 20569.914,E2 20569.914} C_VEL
LIN {X 0,Y 361.456,Z 1137.077,A -85,B 0,C 180,E1 20574.394,E2 20574.394} C_VEL
LIN {X 0,Y 349.344,Z 1162.01,A -85,B 0,C 180,E1 20579.634,E2 20579.634} C_VEL
LIN {X 0,Y 339.612,Z 1182.064,A -85,B 0,C 180,E1 20585.625,E2 20585.625} C_VEL
LIN {X 0,Y 332.503,Z 1197.904,A -85,B 0,C 180,E1 20592.649,E2 20592.649} C_VEL
LIN {X 0,Y 329.058,Z 1207.324,A -85,B 0,C 180,E1 20599.386,E2 20599.386} C_VEL
LIN {X 0,Y 328.015,Z 1211.437,A -85,B 0,C 180,E1 20604.699,E2 20604.699} C_VEL
LIN {X 0,Y 327.896,Z 1212.768,A -85,B 0,C 180,E1 20610,E2 20610} C_VEL
LIN {X 0,Y 328.033,Z 1211.364,A -85,B 0,C 180,E1 20615.301,E2 20615.301} C_VEL
LIN {X 0,Y 329.603,Z 1205.703,A -85,B 0,C 180,E1 20621.94,E2 20621.94} C_VEL
LIN {X 0,Y 334.013,Z 1194.111,A -85,B 0,C 180,E1 20629.203,E2 20629.203} C_VEL
LIN {X 0,Y 341.426,Z 1178.004,A -85,B 0,C 180,E1 20635.641,E2 20635.641} C_VEL
LIN {X 0,Y 351.841,Z 1156.844,A -85,B 0,C 180,E1 20641.48,E2 20641.48} C_VEL
LIN {X 0,Y 363.827,Z 1131.752,A -85,B 0,C 180,E1 20646.406,E2 20646.406} C_VEL
LIN {X 0,Y 376.915,Z 1101.896,A -85,B 0,C 180,E1 20650.601,E2 20650.601} C_VEL
LIN {X 0,Y 389.855,Z 1067.673,A -85,B 0,C 180,E1 20654.003,E2 20654.003} C_VEL
LIN {X 0,Y 401.387,Z 1029.73,A -85,B 0,C 180,E1 20656.612,E2 20656.612} C_VEL
LIN {X 0,Y 408.893,Z 996.668,A -85,B 0,C 180,E1 20658.178,E2 20658.178} C_VEL
LIN {X 0,Y 397.738,Z 966.719,A -85,B 0,C 180,E1 20662.199,E2 20662.199} C_VEL
LIN {X 0,Y 383.32,Z 938.87,A -85,B 0,C 180,E1 20666.848,E2 20666.848} C_VEL
LIN {X 0,Y 368.011,Z 914.88,A -85,B 0,C 180,E1 20672.325,E2 20672.325} C_VEL
LIN {X 0,Y 357.943,Z 900.883,A -85,B 0,C 180,E1 20676.875,E2 20676.875} C_VEL
LIN {X 0,Y 353.923,Z 895.281,A -85,B 0,C 180,E1 20679.079,E2 20679.079} C_VEL
LIN {X 0,Y 349.549,Z 889.115,A -85,B 0,C 180,E1 20681.926,E2 20681.926} C_VEL
LIN {X 0,Y 345.458,Z 882.76,A -85,B 0,C 180,E1 20685.296,E2 20685.296} C_VEL
LIN {X 0,Y 340.575,Z 876.491,A -85,B 0,C 180,E1 20691.531,E2 20691.531} C_VEL
LIN {X 0,Y 340.319,Z 874.897,A -85,B 0,C 180,E1 20692.425,E2 20692.425} C_VEL
LIN {X 0,Y 340.813,Z 875.435,A -85,B 0,C 180,E1 20702.551,E2 20702.551} C_VEL
LIN {X 0,Y 344.062,Z 881.456,A -85,B 0,C 180,E1 20707.276,E2 20707.276} C_VEL
LIN {X 0,Y 346.1,Z 883.685,A -85,B 0,C 180,E1 20709.212,E2 20709.212} C_VEL
LIN {X 0,Y 351.582,Z 891.569,A -85,B 0,C 180,E1 20713.395,E2 20713.395} C_VEL
LIN {X 0,Y 357.356,Z 899.789,A -85,B 0,C 180,E1 20716.789,E2 20716.789} C_VEL
LIN {X 0,Y 366.064,Z 912.41,A -85,B 0,C 180,E1 20720.915,E2 20720.915} C_VEL
LIN {X 0,Y 379.172,Z 933.203,A -85,B 0,C 180,E1 20725.994,E2 20725.994} C_VEL
LIN {X 0,Y 391.814,Z 958.442,A -85,B 0,C 180,E1 20730.634,E2 20730.634} C_VEL
LIN {X 0,Y 402.355,Z 987.3,A -85,B 0,C 180,E1 20734.895,E2 20734.895} C_VEL
LIN {X 0,Y 405.772,Z 999.9,A -85,B 0,C 180,E1 20736.559,E2 20736.559} C_VEL
LIN {X 0,Y 395.422,Z 1041.247,A -85,B 0,C 180,E1 20739.025,E2 20739.025} C_VEL
LIN {X 0,Y 382.962,Z 1080.203,A -85,B 0,C 180,E1 20742.31,E2 20742.31} C_VEL
LIN {X 0,Y 369.308,Z 1116.52,A -85,B 0,C 180,E1 20746.586,E2 20746.586} C_VEL
LIN {X 0,Y 355.439,Z 1149.553,A -85,B 0,C 180,E1 20751.991,E2 20751.991} C_VEL
LIN {X 0,Y 343.615,Z 1177.65,A -85,B 0,C 180,E1 20758.464,E2 20758.464} C_VEL
LIN {X 0,Y 335.051,Z 1199.466,A -85,B 0,C 180,E1 20765.541,E2 20765.541} C_VEL
LIN {X 0,Y 329.882,Z 1215.753,A -85,B 0,C 180,E1 20773.316,E2 20773.316} C_VEL
LIN {X 0,Y 328.073,Z 1225.159,A -85,B 0,C 180,E1 20780.697,E2 20780.697} C_VEL
LIN {X 0,Y 327.745,Z 1229.164,A -85,B 0,C 180,E1 20787.35,E2 20787.35} C_VEL
LIN {X 0,Y 327.739,Z 1229.167,A -85,B 0,C 180,E1 20792.65,E2 20792.65} C_VEL
LIN {X 0,Y 328.039,Z 1225.18,A -85,B 0,C 180,E1 20799.304,E2 20799.304} C_VEL
LIN {X 0,Y 329.916,Z 1215.793,A -85,B 0,C 180,E1 20806.682,E2 20806.682} C_VEL
LIN {X 0,Y 335.037,Z 1199.524,A -85,B 0,C 180,E1 20814.459,E2 20814.459} C_VEL
LIN {X 0,Y 344.18,Z 1176.442,A -85,B 0,C 180,E1 20821.891,E2 20821.891} C_VEL
LIN {X 0,Y 355.927,Z 1148.64,A -85,B 0,C 180,E1 20828.21,E2 20828.21} C_VEL
LIN {X 0,Y 369.726,Z 1115.685,A -85,B 0,C 180,E1 20833.554,E2 20833.554} C_VEL
LIN {X 0,Y 383.754,Z 1078.199,A -85,B 0,C 180,E1 20837.919,E2 20837.919} C_VEL
LIN {X 0,Y 396.779,Z 1037.181,A -85,B 0,C 180,E1 20841.277,E2 20841.277} C_VEL
LIN {X 0,Y 405.942,Z 999.921,A -85,B 0,C 180,E1 20843.449,E2 20843.449} C_VEL
LIN {X 0,Y 396.782,Z 970.327,A -85,B 0,C 180,E1 20847.535,E2 20847.535} C_VEL
LIN {X 0,Y 384.201,Z 942.193,A -85,B 0,C 180,E1 20852.237,E2 20852.237} C_VEL
LIN {X 0,Y 370.671,Z 919.269,A -85,B 0,C 180,E1 20857.3,E2 20857.3} C_VEL
LIN {X 0,Y 364.249,Z 914.539,A -85,B 0,C 180,E1 20859.732,E2 20859.732} C_VEL
LIN {X 0,Y 358.304,Z 910.487,A -85,B 0,C 180,E1 20862.292,E2 20862.292} C_VEL
LIN {X 0,Y 348.222,Z 896.467,A -85,B 0,C 180,E1 20868.389,E2 20868.389} C_VEL
LIN {X 0,Y 343.682,Z 889.721,A -85,B 0,C 180,E1 20872.398,E2 20872.398} C_VEL
LIN {X 0,Y 339.844,Z 883.603,A -85,B 0,C 180,E1 20878.03,E2 20878.03} C_VEL
LIN {X 0,Y 338.743,Z 882.438,A -85,B 0,C 180,E1 20882.56,E2 20882.56} C_VEL
LIN {X 0,Y 339.55,Z 883.658,A -85,B 0,C 180,E1 20887.228,E2 20887.228} C_VEL
LIN {X 0,Y 343.422,Z 889.785,A -85,B 0,C 180,E1 20893.307,E2 20893.307} C_VEL
LIN {X 0,Y 344.994,Z 892.382,A -85,B 0,C 180,E1 20894.92,E2 20894.92} C_VEL
LIN {X 0,Y 349.931,Z 899.107,A -85,B 0,C 180,E1 20898.779,E2 20898.779} C_VEL
LIN {X 0,Y 355.984,Z 907.875,A -85,B 0,C 180,E1 20902.433,E2 20902.433} C_VEL
LIN {X 0,Y 367.096,Z 923.877,A -85,B 0,C 180,E1 20907.577,E2 20907.577} C_VEL
LIN {X 0,Y 381.411,Z 947.157,A -85,B 0,C 180,E1 20912.845,E2 20912.845} C_VEL
LIN {X 0,Y 394.971,Z 975.255,A -85,B 0,C 180,E1 20917.591,E2 20917.591} C_VEL
LIN {X 0,Y 403.566,Z 1000.064,A -85,B 0,C 180,E1 20921.012,E2 20921.012} C_VEL
LIN {X 0,Y 394.033,Z 1037.939,A -85,B 0,C 180,E1 20922.896,E2 20922.896} C_VEL
LIN {X 0,Y 382.106,Z 1074.226,A -85,B 0,C 180,E1 20925.588,E2 20925.588} C_VEL
LIN {X 0,Y 368.892,Z 1107.273,A -85,B 0,C 180,E1 20929.106,E2 20929.106} C_VEL
LIN {X 0,Y 355.101,Z 1137.193,A -85,B 0,C 180,E1 20933.617,E2 20933.617} C_VEL
LIN {X 0,Y 342.329,Z 1162.531,A -85,B 0,C 180,E1 20939.032,E2 20939.032} C_VEL
LIN {X 0,Y 332.328,Z 1182.285,A -85,B 0,C 180,E1 20945.054,E2 20945.054} C_VEL
LIN {X 0,Y 325.088,Z 1197.669,A -85,B 0,C 180,E1 20951.967,E2 20951.967} C_VEL
LIN {X 0,Y 321.258,Z 1207.53,A -85,B 0,C 180,E1 20959.125,E2 20959.125} C_VEL
LIN {X 0,Y 320.123,Z 1211.64,A -85,B 0,C 180,E1 20964.568,E2 20964.568} C_VEL
LIN {X 0,Y 319.996,Z 1212.97,A -85,B 0,C 180,E1 20970,E2 20970} C_VEL
LIN {X 0,Y 320.28,Z 1210.82,A -85,B 0,C 180,E1 20976.68,E2 20976.68} C_VEL
LIN {X 0,Y 322.369,Z 1204.234,A -85,B 0,C 180,E1 20983.593,E2 20983.593} C_VEL
LIN {X 0,Y 327.751,Z 1191.555,A -85,B 0,C 180,E1 20990.997,E2 20990.997} C_VEL
LIN {X 0,Y 336.232,Z 1174.343,A -85,B 0,C 180,E1 20997.512,E2 20997.512} C_VEL
LIN {X 0,Y 347.681,Z 1151.856,A -85,B 0,C 180,E1 21003.383,E2 21003.383} C_VEL
LIN {X 0,Y 361.569,Z 1123.32,A -85,B 0,C 180,E1 21008.565,E2 21008.565} C_VEL
LIN {X 0,Y 375.205,Z 1091.972,A -85,B 0,C 180,E1 21012.568,E2 21012.568} C_VEL
LIN {X 0,Y 388.44,Z 1055.824,A -85,B 0,C 180,E1 21015.792,E2 21015.792} C_VEL
LIN {X 0,Y 399.434,Z 1017.435,A -85,B 0,C 180,E1 21018.126,E2 21018.126} C_VEL
LIN {X 0,Y 403.115,Z 998.961,A -85,B 0,C 180,E1 21019.019,E2 21019.019} C_VEL
LIN {X 0,Y 392.186,Z 969.106,A -85,B 0,C 180,E1 21023.226,E2 21023.226} C_VEL
LIN {X 0,Y 378.409,Z 942.083,A -85,B 0,C 180,E1 21028.011,E2 21028.011} C_VEL
LIN {X 0,Y 365.017,Z 920.877,A -85,B 0,C 180,E1 21033.091,E2 21033.091} C_VEL
LIN {X 0,Y 353.282,Z 903.648,A -85,B 0,C 180,E1 21038.875,E2 21038.875} C_VEL
LIN {X 0,Y 347.599,Z 896.274,A -85,B 0,C 180,E1 21042.585,E2 21042.585} C_VEL
LIN {X 0,Y 343.239,Z 889.745,A -85,B 0,C 180,E1 21046.442,E2 21046.442} C_VEL
LIN {X 0,Y 339.408,Z 883.696,A -85,B 0,C 180,E1 21052.067,E2 21052.067} C_VEL
LIN {X 0,Y 338.584,Z 882.466,A -85,B 0,C 180,E1 21054.87,E2 21054.87} C_VEL
LIN {X 0,Y 339.723,Z 883.43,A -85,B 0,C 180,E1 21062.399,E2 21062.399} C_VEL
LIN {X 0,Y 343.242,Z 889.484,A -85,B 0,C 180,E1 21067.453,E2 21067.453} C_VEL
LIN {X 0,Y 344.869,Z 891.698,A -85,B 0,C 180,E1 21069.056,E2 21069.056} C_VEL
LIN {X 0,Y 350.097,Z 899.321,A -85,B 0,C 180,E1 21073.134,E2 21073.134} C_VEL
LIN {X 0,Y 358.461,Z 910.995,A -85,B 0,C 180,E1 21077.925,E2 21077.925} C_VEL
LIN {X 0,Y 371.101,Z 931.145,A -85,B 0,C 180,E1 21083.543,E2 21083.543} C_VEL
LIN {X 0,Y 383.353,Z 954.165,A -85,B 0,C 180,E1 21088.361,E2 21088.361} C_VEL
LIN {X 0,Y 394.189,Z 981.468,A -85,B 0,C 180,E1 21092.823,E2 21092.823} C_VEL
LIN {X 0,Y 399.993,Z 1004.117,A -85,B 0,C 180,E1 21095.911,E2 21095.911} C_VEL
LIN {X 0,Y 389.608,Z 1043.19,A -85,B 0,C 180,E1 21098.289,E2 21098.289} C_VEL
LIN {X 0,Y 377.165,Z 1080.783,A -85,B 0,C 180,E1 21101.505,E2 21101.505} C_VEL
LIN {X 0,Y 363.452,Z 1116.176,A -85,B 0,C 180,E1 21105.706,E2 21105.706} C_VEL
LIN {X 0,Y 349.358,Z 1148.607,A -85,B 0,C 180,E1 21111.036,E2 21111.036} C_VEL
LIN {X 0,Y 336.741,Z 1177.141,A -85,B 0,C 180,E1 21117.657,E2 21117.657} C_VEL
LIN {X 0,Y 327.65,Z 1199.235,A -85,B 0,C 180,E1 21124.951,E2 21124.951} C_VEL
LIN {X 0,Y 322.186,Z 1215.534,A -85,B 0,C 180,E1 21132.905,E2 21132.905} C_VEL
LIN {X 0,Y 320.186,Z 1224.951,A -85,B 0,C 180,E1 21140.465,E2 21140.465} C_VEL
LIN {X 0,Y 319.835,Z 1228.962,A -85,B 0,C 180,E1 21147.284,E2 21147.284} C_VEL
LIN {X 0,Y 319.83,Z 1228.965,A -85,B 0,C 180,E1 21152.715,E2 21152.715} C_VEL
LIN {X 0,Y 320.155,Z 1224.973,A -85,B 0,C 180,E1 21159.535,E2 21159.535} C_VEL
LIN {X 0,Y 322.216,Z 1215.577,A -85,B 0,C 180,E1 21167.092,E2 21167.092} C_VEL
LIN {X 0,Y 327.64,Z 1199.296,A -85,B 0,C 180,E1 21175.049,E2 21175.049} C_VEL
LIN {X 0,Y 337.169,Z 1176.177,A -85,B 0,C 180,E1 21182.636,E2 21182.636} C_VEL
LIN {X 0,Y 349.398,Z 1148.734,A -85,B 0,C 180,E1 21188.96,E2 21188.96} C_VEL
LIN {X 0,Y 363.857,Z 1115.323,A -85,B 0,C 180,E1 21194.44,E2 21194.44} C_VEL
LIN {X 0,Y 378.38,Z 1077.662,A -85,B 0,C 180,E1 21198.837,E2 21198.837} C_VEL
LIN {X 0,Y 391.834,Z 1036.259,A -85,B 0,C 180,E1 21202.216,E2 21202.216} C_VEL
LIN {X 0,Y 400.281,Z 1002.7,A -85,B 0,C 180,E1 21204.207,E2 21204.207} C_VEL
LIN {X 0,Y 391.465,Z 973.314,A -85,B 0,C 180,E1 21208.431,E2 21208.431} C_VEL
LIN {X 0,Y 379.663,Z 946.403,A -85,B 0,C 180,E1 21213.164,E2 21213.164} C_VEL
LIN {X 0,Y 366.969,Z 924.206,A -85,B 0,C 180,E1 21218.266,E2 21218.266} C_VEL
LIN {X 0,Y 358.304,Z 910.487,A -85,B 0,C 180,E1 21222.292,E2 21222.292} C_VEL
LIN {X 0,Y 354.455,Z 909.704,A -85,B 0,C 180,E1 21224.062,E2 21224.062} C_VEL
LIN {X 0,Y 350.702,Z 910.039,A -85,B 0,C 180,E1 21225.92,E2 21225.92} C_VEL
LIN {X 0,Y 346.398,Z 903.686,A -85,B 0,C 180,E1 21228.966,E2 21228.966} C_VEL
LIN {X 0,Y 342.424,Z 897.412,A -85,B 0,C 180,E1 21232.656,E2 21232.656} C_VEL
LIN {X 0,Y 338.725,Z 891.122,A -85,B 0,C 180,E1 21238.392,E2 21238.392} C_VEL
LIN {X 0,Y 338.444,Z 890.901,A -85,B 0,C 180,E1 21246.714,E2 21246.714} C_VEL
LIN {X 0,Y 341.775,Z 897.205,A -85,B 0,C 180,E1 21252.597,E2 21252.597} C_VEL
LIN {X 0,Y 343.482,Z 899.518,A -85,B 0,C 180,E1 21254.406,E2 21254.406} C_VEL
LIN {X 0,Y 348.642,Z 907.069,A -85,B 0,C 180,E1 21258.605,E2 21258.605} C_VEL
LIN {X 0,Y 356.486,Z 918.04,A -85,B 0,C 180,E1 21263.225,E2 21263.225} C_VEL
LIN {X 0,Y 368.913,Z 937.495,A -85,B 0,C 180,E1 21268.805,E2 21268.805} C_VEL
LIN {X 0,Y 381.551,Z 960.189,A -85,B 0,C 180,E1 21273.596,E2 21273.596} C_VEL
LIN {X 0,Y 393.4,Z 988.258,A -85,B 0,C 180,E1 21278.172,E2 21278.172} C_VEL
LIN {X 0,Y 397.832,Z 1004.039,A -85,B 0,C 180,E1 21280.274,E2 21280.274} C_VEL
LIN {X 0,Y 387.167,Z 1043.875,A -85,B 0,C 180,E1 21282.377,E2 21282.377} C_VEL
LIN {X 0,Y 373.617,Z 1082.281,A -85,B 0,C 180,E1 21285.447,E2 21285.447} C_VEL
LIN {X 0,Y 359.051,Z 1116.106,A -85,B 0,C 180,E1 21289.41,E2 21289.41} C_VEL
LIN {X 0,Y 345.062,Z 1144.638,A -85,B 0,C 180,E1 21294.189,E2 21294.189} C_VEL
LIN {X 0,Y 331.975,Z 1169.3,A -85,B 0,C 180,E1 21300.107,E2 21300.107} C_VEL
LIN {X 0,Y 321.902,Z 1188.705,A -85,B 0,C 180,E1 21306.967,E2 21306.967} C_VEL
LIN {X 0,Y 315.333,Z 1202.825,A -85,B 0,C 180,E1 21314.725,E2 21314.725} C_VEL
LIN {X 0,Y 312.665,Z 1210.143,A -85,B 0,C 180,E1 21321.64,E2 21321.64} C_VEL
LIN {X 0,Y 312.044,Z 1212.853,A -85,B 0,C 180,E1 21327.217,E2 21327.217} C_VEL
LIN {X 0,Y 312.086,Z 1212.812,A -85,B 0,C 180,E1 21332.783,E2 21332.783} C_VEL
LIN {X 0,Y 313.104,Z 1208.89,A -85,B 0,C 180,E1 21339.752,E2 21339.752} C_VEL
LIN {X 0,Y 316.774,Z 1199.424,A -85,B 0,C 180,E1 21347.396,E2 21347.396} C_VEL
LIN {X 0,Y 323.42,Z 1185.552,A -85,B 0,C 180,E1 21354.215,E2 21354.215} C_VEL
LIN {X 0,Y 333.758,Z 1165.886,A -85,B 0,C 180,E1 21360.715,E2 21360.715} C_VEL
LIN {X 0,Y 346.44,Z 1141.632,A -85,B 0,C 180,E1 21366.276,E2 21366.276} C_VEL
LIN {X 0,Y 360.408,Z 1112.855,A -85,B 0,C 180,E1 21370.922,E2 21370.922} C_VEL
LIN {X 0,Y 374.147,Z 1080.481,A -85,B 0,C 180,E1 21374.617,E2 21374.617} C_VEL
LIN {X 0,Y 387.345,Z 1042.669,A -85,B 0,C 180,E1 21377.595,E2 21377.595} C_VEL
LIN {X 0,Y 397.749,Z 1003.423,A -85,B 0,C 180,E1 21379.653,E2 21379.653} C_VEL
LIN {X 0,Y 388.918,Z 976.612,A -85,B 0,C 180,E1 21383.475,E2 21383.475} C_VEL
LIN {X 0,Y 376.135,Z 949.818,A -85,B 0,C 180,E1 21388.258,E2 21388.258} C_VEL
LIN {X 0,Y 362.797,Z 927.842,A -85,B 0,C 180,E1 21393.564,E2 21393.564} C_VEL
LIN {X 0,Y 351.449,Z 910.908,A -85,B 0,C 180,E1 21399.338,E2 21399.338} C_VEL
LIN {X 0,Y 346.062,Z 903.733,A -85,B 0,C 180,E1 21402.981,E2 21402.981} C_VEL
LIN {X 0,Y 341.869,Z 897.365,A -85,B 0,C 180,E1 21406.839,E2 21406.839} C_VEL
LIN {X 0,Y 338.311,Z 891.182,A -85,B 0,C 180,E1 21412.437,E2 21412.437} C_VEL
LIN {X 0,Y 338.569,Z 890.727,A -85,B 0,C 180,E1 21421.927,E2 21421.927} C_VEL
LIN {X 0,Y 341.952,Z 897.123,A -85,B 0,C 180,E1 21427.161,E2 21427.161} C_VEL
LIN {X 0,Y 343.656,Z 899.705,A -85,B 0,C 180,E1 21428.91,E2 21428.91} C_VEL
LIN {X 0,Y 348.628,Z 907,A -85,B 0,C 180,E1 21432.871,E2 21432.871} C_VEL
LIN {X 0,Y 356.699,Z 918.599,A -85,B 0,C 180,E1 21437.617,E2 21437.617} C_VEL
LIN {X 0,Y 369.567,Z 939.873,A -85,B 0,C 180,E1 21443.591,E2 21443.591} C_VEL
LIN {X 0,Y 381.531,Z 964.595,A -85,B 0,C 180,E1 21448.647,E2 21448.647} C_VEL
LIN {X 0,Y 391.213,Z 992.534,A -85,B 0,C 180,E1 21453.162,E2 21453.162} C_VEL
LIN {X 0,Y 394.34,Z 1007.615,A -85,B 0,C 180,E1 21455.19,E2 21455.19} C_VEL
LIN {X 0,Y 382.339,Z 1050.186,A -85,B 0,C 180,E1 21457.911,E2 21457.911} C_VEL
LIN {X 0,Y 368.291,Z 1089.5,A -85,B 0,C 180,E1 21461.522,E2 21461.522} C_VEL
LIN {X 0,Y 354.15,Z 1123.704,A -85,B 0,C 180,E1 21465.95,E2 21465.95} C_VEL
LIN {X 0,Y 340.911,Z 1152.669,A -85,B 0,C 180,E1 21471.069,E2 21471.069} C_VEL
LIN {X 0,Y 329.244,Z 1178.141,A -85,B 0,C 180,E1 21477.263,E2 21477.263} C_VEL
LIN {X 0,Y 319.84,Z 1200.003,A -85,B 0,C 180,E1 21484.761,E2 21484.761} C_VEL
LIN {X 0,Y 314.473,Z 1215.315,A -85,B 0,C 180,E1 21492.473,E2 21492.473} C_VEL
LIN {X 0,Y 312.312,Z 1224.744,A -85,B 0,C 180,E1 21500.223,E2 21500.223} C_VEL
LIN {X 0,Y 311.95,Z 1228.76,A -85,B 0,C 180,E1 21507.215,E2 21507.215} C_VEL
LIN {X 0,Y 311.946,Z 1228.764,A -85,B 0,C 180,E1 21512.784,E2 21512.784} C_VEL
LIN {X 0,Y 312.285,Z 1224.767,A -85,B 0,C 180,E1 21519.778,E2 21519.778} C_VEL
LIN {X 0,Y 314.498,Z 1215.36,A -85,B 0,C 180,E1 21527.525,E2 21527.525} C_VEL
LIN {X 0,Y 320.28,Z 1198.949,A -85,B 0,C 180,E1 21535.717,E2 21535.717} C_VEL
LIN {X 0,Y 329.746,Z 1177.103,A -85,B 0,C 180,E1 21543.072,E2 21543.072} C_VEL
LIN {X 0,Y 342.849,Z 1148.941,A -85,B 0,C 180,E1 21549.719,E2 21549.719} C_VEL
LIN {X 0,Y 357.632,Z 1116.007,A -85,B 0,C 180,E1 21555.21,E2 21555.21} C_VEL
LIN {X 0,Y 372.828,Z 1077.943,A -85,B 0,C 180,E1 21559.702,E2 21559.702} C_VEL
LIN {X 0,Y 386.387,Z 1037.505,A -85,B 0,C 180,E1 21563.039,E2 21563.039} C_VEL
LIN {X 0,Y 394.613,Z 1005.445,A -85,B 0,C 180,E1 21565.006,E2 21565.006} C_VEL
LIN {X 0,Y 386.487,Z 977.277,A -85,B 0,C 180,E1 21569.221,E2 21569.221} C_VEL
LIN {X 0,Y 375.831,Z 951.843,A -85,B 0,C 180,E1 21573.848,E2 21573.848} C_VEL
LIN {X 0,Y 363.389,Z 929.033,A -85,B 0,C 180,E1 21579.243,E2 21579.243} C_VEL
LIN {X 0,Y 353.53,Z 914.082,A -85,B 0,C 180,E1 21584.223,E2 21584.223} C_VEL
LIN {X 0,Y 350.702,Z 910.039,A -85,B 0,C 180,E1 21585.92,E2 21585.92} C_VEL
LIN {X 0,Y 344.43,Z 910.708,A -85,B 0,C 180,E1 21589.687,E2 21589.687} C_VEL
LIN {X 0,Y 340.828,Z 904.846,A -85,B 0,C 180,E1 21593.283,E2 21593.283} C_VEL
LIN {X 0,Y 337.464,Z 898.276,A -85,B 0,C 180,E1 21599.302,E2 21599.302} C_VEL
LIN {X 0,Y 337.458,Z 899.241,A -85,B 0,C 180,E1 21606.811,E2 21606.811} C_VEL
LIN {X 0,Y 341.289,Z 905.38,A -85,B 0,C 180,E1 21613.099,E2 21613.099} C_VEL
LIN {X 0,Y 347.474,Z 915.11,A -85,B 0,C 180,E1 21618.505,E2 21618.505} C_VEL
LIN {X 0,Y 354.962,Z 925.999,A -85,B 0,C 180,E1 21622.999,E2 21622.999} C_VEL
LIN {X 0,Y 366.332,Z 944.255,A -85,B 0,C 180,E1 21628.311,E2 21628.311} C_VEL
LIN {X 0,Y 378.255,Z 966.984,A -85,B 0,C 180,E1 21633.204,E2 21633.204} C_VEL
LIN {X 0,Y 388.839,Z 993.568,A -85,B 0,C 180,E1 21637.642,E2 21637.642} C_VEL
LIN {X 0,Y 392.509,Z 1006.285,A -85,B 0,C 180,E1 21639.457,E2 21639.457} C_VEL
LIN {X 0,Y 381.341,Z 1046.237,A -85,B 0,C 180,E1 21641.623,E2 21641.623} C_VEL
LIN {X 0,Y 367.748,Z 1083.316,A -85,B 0,C 180,E1 21644.646,E2 21644.646} C_VEL
LIN {X 0,Y 353.043,Z 1116.423,A -85,B 0,C 180,E1 21648.57,E2 21648.57} C_VEL
LIN {X 0,Y 338.154,Z 1145.754,A -85,B 0,C 180,E1 21653.579,E2 21653.579} C_VEL
LIN {X 0,Y 324.588,Z 1170.341,A -85,B 0,C 180,E1 21659.652,E2 21659.652} C_VEL
LIN {X 0,Y 314.258,Z 1189.437,A -85,B 0,C 180,E1 21666.635,E2 21666.635} C_VEL
LIN {X 0,Y 308.296,Z 1201.6,A -85,B 0,C 180,E1 21673.301,E2 21673.301} C_VEL
LIN {X 0,Y 304.826,Z 1210.347,A -85,B 0,C 180,E1 21681.424,E2 21681.424} C_VEL
LIN {X 0,Y 304.144,Z 1213.055,A -85,B 0,C 180,E1 21687.145,E2 21687.145} C_VEL
LIN {X 0,Y 304.185,Z 1213.014,A -85,B 0,C 180,E1 21692.856,E2 21692.856} C_VEL
LIN {X 0,Y 305.291,Z 1209.095,A -85,B 0,C 180,E1 21700.005,E2 21700.005} C_VEL
LIN {X 0,Y 309.148,Z 1199.637,A -85,B 0,C 180,E1 21707.839,E2 21707.839} C_VEL
LIN {X 0,Y 316.455,Z 1185.189,A -85,B 0,C 180,E1 21715.047,E2 21715.047} C_VEL
LIN {X 0,Y 327.579,Z 1164.964,A -85,B 0,C 180,E1 21721.748,E2 21721.748} C_VEL
LIN {X 0,Y 340.721,Z 1140.634,A -85,B 0,C 180,E1 21727.313,E2 21727.313} C_VEL
LIN {X 0,Y 355.159,Z 1111.618,A -85,B 0,C 180,E1 21731.975,E2 21731.975} C_VEL
LIN {X 0,Y 368.992,Z 1079.779,A -85,B 0,C 180,E1 21735.59,E2 21735.59} C_VEL
LIN {X 0,Y 382.094,Z 1043.324,A -85,B 0,C 180,E1 21738.464,E2 21738.464} C_VEL
LIN {X 0,Y 392.27,Z 1006.435,A -85,B 0,C 180,E1 21740.436,E2 21740.436} C_VEL
LIN {X 0,Y 383.743,Z 979.894,A -85,B 0,C 180,E1 21744.393,E2 21744.393} C_VEL
LIN {X 0,Y 371.482,Z 953.413,A -85,B 0,C 180,E1 21749.362,E2 21749.362} C_VEL
LIN {X 0,Y 359.326,Z 932.902,A -85,B 0,C 180,E1 21754.61,E2 21754.61} C_VEL
LIN {X 0,Y 349.392,Z 917.898,A -85,B 0,C 180,E1 21759.956,E2 21759.956} C_VEL
LIN {X 0,Y 344.328,Z 910.916,A -85,B 0,C 180,E1 21763.551,E2 21763.551} C_VEL
LIN {X 0,Y 340.596,Z 905.048,A -85,B 0,C 180,E1 21767.154,E2 21767.154} C_VEL
LIN {X 0,Y 337.214,Z 898.58,A -85,B 0,C 180,E1 21772.874,E2 21772.874} C_VEL
LIN {X 0,Y 337.531,Z 898.859,A -85,B 0,C 180,E1 21781.852,E2 21781.852} C_VEL
LIN {X 0,Y 341.123,Z 905.127,A -85,B 0,C 180,E1 21787.339,E2 21787.339} C_VEL
LIN {X 0,Y 347.06,Z 914.509,A -85,B 0,C 180,E1 21792.529,E2 21792.529} C_VEL
LIN {X 0,Y 354.601,Z 925.714,A -85,B 0,C 180,E1 21797.164,E2 21797.164} C_VEL
LIN {X 0,Y 366.153,Z 945.792,A -85,B 0,C 180,E1 21802.916,E2 21802.916} C_VEL
LIN {X 0,Y 377.096,Z 969.371,A -85,B 0,C 180,E1 21807.929,E2 21807.929} C_VEL
LIN {X 0,Y 386.355,Z 997.564,A -85,B 0,C 180,E1 21812.628,E2 21812.628} C_VEL
LIN {X 0,Y 388.998,Z 1009.819,A -85,B 0,C 180,E1 21814.378,E2 21814.378} C_VEL
LIN {X 0,Y 376.757,Z 1051.685,A -85,B 0,C 180,E1 21817.098,E2 21817.098} C_VEL
LIN {X 0,Y 361.813,Z 1091.972,A -85,B 0,C 180,E1 21820.877,E2 21820.877} C_VEL
LIN {X 0,Y 346.56,Z 1127.28,A -85,B 0,C 180,E1 21825.606,E2 21825.606} C_VEL
LIN {X 0,Y 331.687,Z 1158.533,A -85,B 0,C 180,E1 21831.504,E2 21831.504} C_VEL
LIN {X 0,Y 319.283,Z 1184.63,A -85,B 0,C 180,E1 21838.53,E2 21838.53} C_VEL
LIN {X 0,Y 310.494,Z 1204.575,A -85,B 0,C 180,E1 21846.257,E2 21846.257} C_VEL
LIN {X 0,Y 305.674,Z 1218.972,A -85,B 0,C 180,E1 21854.754,E2 21854.754} C_VEL
LIN {X 0,Y 304.289,Z 1225.725,A -85,B 0,C 180,E1 21861.408,E2 21861.408} C_VEL
LIN {X 0,Y 304.039,Z 1228.558,A -85,B 0,C 180,E1 21867.143,E2 21867.143} C_VEL
LIN {X 0,Y 304.037,Z 1228.562,A -85,B 0,C 180,E1 21872.856,E2 21872.856} C_VEL
LIN {X 0,Y 304.42,Z 1224.56,A -85,B 0,C 180,E1 21880.033,E2 21880.033} C_VEL
LIN {X 0,Y 306.787,Z 1215.143,A -85,B 0,C 180,E1 21887.981,E2 21887.981} C_VEL
LIN {X 0,Y 312.975,Z 1198.719,A -85,B 0,C 180,E1 21896.363,E2 21896.363} C_VEL
LIN {X 0,Y 322.897,Z 1176.856,A -85,B 0,C 180,E1 21903.867,E2 21903.867} C_VEL
LIN {X 0,Y 336.58,Z 1148.765,A -85,B 0,C 180,E1 21910.582,E2 21910.582} C_VEL
LIN {X 0,Y 351.907,Z 1115.655,A -85,B 0,C 180,E1 21916.157,E2 21916.157} C_VEL
LIN {X 0,Y 367.616,Z 1077.521,A -85,B 0,C 180,E1 21920.661,E2 21920.661} C_VEL
LIN {X 0,Y 381.574,Z 1036.836,A -85,B 0,C 180,E1 21924.01,E2 21924.01} C_VEL
LIN {X 0,Y 389.24,Z 1009.099,A -85,B 0,C 180,E1 21925.697,E2 21925.697} C_VEL
LIN {X 0,Y 381.816,Z 981.933,A -85,B 0,C 180,E1 21929.897,E2 21929.897} C_VEL
LIN {X 0,Y 371.759,Z 956.804,A -85,B 0,C 180,E1 21934.612,E2 21934.612} C_VEL
LIN {X 0,Y 360.2,Z 934.933,A -85,B 0,C 180,E1 21940.065,E2 21940.065} C_VEL
LIN {X 0,Y 350.192,Z 918.613,A -85,B 0,C 180,E1 21945.594,E2 21945.594} C_VEL
LIN {X 0,Y 344.604,Z 910.886,A -85,B 0,C 180,E1 21949.549,E2 21949.549} C_VEL
LIN {X 0,Y 344.43,Z 910.708,A -85,B 0,C 180,E1 21949.687,E2 21949.687} C_VEL
LIN {X 0,Y 341.86,Z 911.289,A -85,B 0,C 180,E1 21951.604,E2 21951.604} C_VEL
LIN {X 0,Y 339.581,Z 912.522,A -85,B 0,C 180,E1 21953.562,E2 21953.562} C_VEL
LIN {X 0,Y 336.281,Z 906.013,A -85,B 0,C 180,E1 21959.996,E2 21959.996} C_VEL
LIN {X 0,Y 336.421,Z 907.008,A -85,B 0,C 180,E1 21966.6,E2 21966.6} C_VEL
LIN {X 0,Y 340.993,Z 914.901,A -85,B 0,C 180,E1 21973.893,E2 21973.893} C_VEL
LIN {X 0,Y 345.991,Z 922.615,A -85,B 0,C 180,E1 21978.174,E2 21978.174} C_VEL
LIN {X 0,Y 353.362,Z 933.741,A -85,B 0,C 180,E1 21982.752,E2 21982.752} C_VEL
LIN {X 0,Y 364.561,Z 952.628,A -85,B 0,C 180,E1 21988.264,E2 21988.264} C_VEL
LIN {X 0,Y 375.868,Z 975.921,A -85,B 0,C 180,E1 21993.218,E2 21993.218} C_VEL
LIN {X 0,Y 385.54,Z 1003.369,A -85,B 0,C 180,E1 21997.791,E2 21997.791} C_VEL
LIN {X 0,Y 386.715,Z 1010.418,A -85,B 0,C 180,E1 21998.704,E2 21998.704} C_VEL
LIN {X 0,Y 375.585,Z 1048.489,A -85,B 0,C 180,E1 22000.847,E2 22000.847} C_VEL
LIN {X 0,Y 362.122,Z 1083.982,A -85,B 0,C 180,E1 22003.783,E2 22003.783} C_VEL
LIN {X 0,Y 347.081,Z 1116.811,A -85,B 0,C 180,E1 22007.712,E2 22007.712} C_VEL
LIN {X 0,Y 331.777,Z 1146.011,A -85,B 0,C 180,E1 22012.761,E2 22012.761} C_VEL
LIN {X 0,Y 318.667,Z 1169.076,A -85,B 0,C 180,E1 22018.463,E2 22018.463} C_VEL
LIN {X 0,Y 307.702,Z 1188.31,A -85,B 0,C 180,E1 22025.41,E2 22025.41} C_VEL
LIN {X 0,Y 300.285,Z 1202.609,A -85,B 0,C 180,E1 22033.426,E2 22033.426} C_VEL
LIN {X 0,Y 296.97,Z 1210.551,A -85,B 0,C 180,E1 22041.195,E2 22041.195} C_VEL
LIN {X 0,Y 296.263,Z 1213.257,A -85,B 0,C 180,E1 22047.069,E2 22047.069} C_VEL
LIN {X 0,Y 296.302,Z 1213.217,A -85,B 0,C 180,E1 22052.932,E2 22052.932} C_VEL
LIN {X 0,Y 297.459,Z 1209.3,A -85,B 0,C 180,E1 22060.271,E2 22060.271} C_VEL
LIN {X 0,Y 301.539,Z 1199.847,A -85,B 0,C 180,E1 22068.305,E2 22068.305} C_VEL
LIN {X 0,Y 308.813,Z 1186.13,A -85,B 0,C 180,E1 22075.379,E2 22075.379} C_VEL
LIN {X 0,Y 320.147,Z 1166.381,A -85,B 0,C 180,E1 22082.173,E2 22082.173} C_VEL
LIN {X 0,Y 333.559,Z 1142.542,A -85,B 0,C 180,E1 22087.827,E2 22087.827} C_VEL
LIN {X 0,Y 348.495,Z 1113.671,A -85,B 0,C 180,E1 22092.619,E2 22092.619} C_VEL
LIN {X 0,Y 363.735,Z 1079.655,A -85,B 0,C 180,E1 22096.533,E2 22096.533} C_VEL
LIN {X 0,Y 377.489,Z 1042.095,A -85,B 0,C 180,E1 22099.48,E2 22099.48} C_VEL
LIN {X 0,Y 386.687,Z 1008.077,A -85,B 0,C 180,E1 22101.386,E2 22101.386} C_VEL
LIN {X 0,Y 377.734,Z 980.693,A -85,B 0,C 180,E1 22105.76,E2 22105.76} C_VEL
LIN {X 0,Y 366.209,Z 955.968,A -85,B 0,C 180,E1 22110.798,E2 22110.798} C_VEL
LIN {X 0,Y 355.172,Z 936.785,A -85,B 0,C 180,E1 22116.042,E2 22116.042} C_VEL
LIN {X 0,Y 346.918,Z 924.246,A -85,B 0,C 180,E1 22120.886,E2 22120.886} C_VEL
LIN {X 0,Y 342.913,Z 918.423,A -85,B 0,C 180,E1 22123.893,E2 22123.893} C_VEL
LIN {X 0,Y 339.373,Z 912.708,A -85,B 0,C 180,E1 22127.435,E2 22127.435} C_VEL
LIN {X 0,Y 336.04,Z 906.14,A -85,B 0,C 180,E1 22133.531,E2 22133.531} C_VEL
LIN {X 0,Y 336.484,Z 906.755,A -85,B 0,C 180,E1 22141.697,E2 22141.697} C_VEL
LIN {X 0,Y 340.886,Z 914.717,A -85,B 0,C 180,E1 22148.215,E2 22148.215} C_VEL
LIN {X 0,Y 346.024,Z 922.887,A -85,B 0,C 180,E1 22152.568,E2 22152.568} C_VEL
LIN {X 0,Y 352.968,Z 933.739,A -85,B 0,C 180,E1 22157.004,E2 22157.004} C_VEL
LIN {X 0,Y 363.602,Z 953.202,A -85,B 0,C 180,E1 22162.643,E2 22162.643} C_VEL
LIN {X 0,Y 373.852,Z 977.178,A -85,B 0,C 180,E1 22167.772,E2 22167.772} C_VEL
LIN {X 0,Y 382.029,Z 1004.934,A -85,B 0,C 180,E1 22172.458,E2 22172.458} C_VEL
LIN {X 0,Y 383.576,Z 1012.373,A -85,B 0,C 180,E1 22173.571,E2 22173.571} C_VEL
LIN {X 0,Y 371.568,Z 1052.134,A -85,B 0,C 180,E1 22176.18,E2 22176.18} C_VEL
LIN {X 0,Y 356.089,Z 1092.59,A -85,B 0,C 180,E1 22180.006,E2 22180.006} C_VEL
LIN {X 0,Y 340.162,Z 1128.185,A -85,B 0,C 180,E1 22184.848,E2 22184.848} C_VEL
LIN {X 0,Y 325.142,Z 1158.611,A -85,B 0,C 180,E1 22190.69,E2 22190.69} C_VEL
LIN {X 0,Y 312.328,Z 1184.385,A -85,B 0,C 180,E1 22197.745,E2 22197.745} C_VEL
LIN {X 0,Y 303.074,Z 1204.346,A -85,B 0,C 180,E1 22205.639,E2 22205.639} C_VEL
LIN {X 0,Y 298.088,Z 1217.966,A -85,B 0,C 180,E1 22213.764,E2 22213.764} C_VEL
LIN {X 0,Y 296.401,Z 1225.52,A -85,B 0,C 180,E1 22221.177,E2 22221.177} C_VEL
LIN {X 0,Y 296.135,Z 1228.356,A -85,B 0,C 180,E1 22227.067,E2 22227.067} C_VEL
LIN {X 0,Y 296.134,Z 1228.36,A -85,B 0,C 180,E1 22232.933,E2 22232.933} C_VEL
LIN {X 0,Y 296.577,Z 1224.355,A -85,B 0,C 180,E1 22240.301,E2 22240.301} C_VEL
LIN {X 0,Y 299.078,Z 1214.926,A -85,B 0,C 180,E1 22248.461,E2 22248.461} C_VEL
LIN {X 0,Y 305.356,Z 1199.185,A -85,B 0,C 180,E1 22256.74,E2 22256.74} C_VEL
LIN {X 0,Y 316.151,Z 1176.612,A -85,B 0,C 180,E1 22264.691,E2 22264.691} C_VEL
LIN {X 0,Y 329.941,Z 1149.39,A -85,B 0,C 180,E1 22271.314,E2 22271.314} C_VEL
LIN {X 0,Y 345.829,Z 1116.314,A -85,B 0,C 180,E1 22276.987,E2 22276.987} C_VEL
LIN {X 0,Y 362.061,Z 1078.276,A -85,B 0,C 180,E1 22281.537,E2 22281.537} C_VEL
LIN {X 0,Y 376.308,Z 1038.088,A -85,B 0,C 180,E1 22284.878,E2 22284.878} C_VEL
LIN {X 0,Y 383.778,Z 1012.278,A -85,B 0,C 180,E1 22286.449,E2 22286.449} C_VEL
LIN {X 0,Y 376.708,Z 985.147,A -85,B 0,C 180,E1 22290.814,E2 22290.814} C_VEL
LIN {X 0,Y 367.083,Z 960.476,A -85,B 0,C 180,E1 22295.704,E2 22295.704} C_VEL
LIN {X 0,Y 356.717,Z 940.183,A -85,B 0,C 180,E1 22301.022,E2 22301.022} C_VEL
LIN {X 0,Y 348.149,Z 925.705,A -85,B 0,C 180,E1 22306.15,E2 22306.15} C_VEL
LIN {X 0,Y 342.867,Z 918.051,A -85,B 0,C 180,E1 22310.138,E2 22310.138} C_VEL
LIN {X 0,Y 339.742,Z 912.623,A -85,B 0,C 180,E1 22313.386,E2 22313.386} C_VEL
LIN {X 0,Y 339.581,Z 912.522,A -85,B 0,C 180,E1 22313.562,E2 22313.562} C_VEL
LIN {X 0,Y 336.162,Z 916.912,A -85,B 0,C 180,E1 22317.227,E2 22317.227} C_VEL
LIN {X 0,Y 336.048,Z 916.695,A -85,B 0,C 180,E1 22317.474,E2 22317.474} C_VEL
LIN {X 0,Y 335.32,Z 913.841,A -85,B 0,C 180,E1 22319.996,E2 22319.996} C_VEL
LIN {X 0,Y 335.389,Z 914.771,A -85,B 0,C 180,E1 22326.388,E2 22326.388} C_VEL
LIN {X 0,Y 339.727,Z 922.59,A -85,B 0,C 180,E1 22333.617,E2 22333.617} C_VEL
LIN {X 0,Y 344.91,Z 930.832,A -85,B 0,C 180,E1 22338.15,E2 22338.15} C_VEL
LIN {X 0,Y 352.114,Z 942.355,A -85,B 0,C 180,E1 22342.777,E2 22342.777} C_VEL
LIN {X 0,Y 362.432,Z 960.653,A -85,B 0,C 180,E1 22348.113,E2 22348.113} C_VEL
LIN {X 0,Y 373.213,Z 985.105,A -85,B 0,C 180,E1 22353.311,E2 22353.311} C_VEL
LIN {X 0,Y 381.564,Z 1011.672,A -85,B 0,C 180,E1 22357.763,E2 22357.763} C_VEL
LIN {X 0,Y 370.474,Z 1049.053,A -85,B 0,C 180,E1 22359.924,E2 22359.924} C_VEL
LIN {X 0,Y 357.04,Z 1083.613,A -85,B 0,C 180,E1 22362.786,E2 22362.786} C_VEL
LIN {X 0,Y 341.314,Z 1116.988,A -85,B 0,C 180,E1 22366.794,E2 22366.794} C_VEL
LIN {X 0,Y 325.484,Z 1146.271,A -85,B 0,C 180,E1 22371.914,E2 22371.914} C_VEL
LIN {X 0,Y 311.871,Z 1169.307,A -85,B 0,C 180,E1 22377.693,E2 22377.693} C_VEL
LIN {X 0,Y 300.581,Z 1188.299,A -85,B 0,C 180,E1 22384.673,E2 22384.673} C_VEL
LIN {X 0,Y 292.629,Z 1202.815,A -85,B 0,C 180,E1 22392.979,E2 22392.979} C_VEL
LIN {X 0,Y 289.138,Z 1210.755,A -85,B 0,C 180,E1 22400.955,E2 22400.955} C_VEL
LIN {X 0,Y 288.382,Z 1213.458,A -85,B 0,C 180,E1 22406.988,E2 22406.988} C_VEL
LIN {X 0,Y 288.406,Z 1213.2,A -85,B 0,C 180,E1 22413.69,E2 22413.69} C_VEL
LIN {X 0,Y 290.134,Z 1208.226,A -85,B 0,C 180,E1 22422.059,E2 22422.059} C_VEL
LIN {X 0,Y 295.201,Z 1197.755,A -85,B 0,C 180,E1 22430.273,E2 22430.273} C_VEL
LIN {X 0,Y 304.743,Z 1181.046,A -85,B 0,C 180,E1 22438.189,E2 22438.189} C_VEL
LIN {X 0,Y 317.687,Z 1159.422,A -85,B 0,C 180,E1 22444.916,E2 22444.916} C_VEL
LIN {X 0,Y 332.634,Z 1133.269,A -85,B 0,C 180,E1 22450.478,E2 22450.478} C_VEL
LIN {X 0,Y 348.281,Z 1102.671,A -85,B 0,C 180,E1 22454.992,E2 22454.992} C_VEL
LIN {X 0,Y 363.265,Z 1068.258,A -85,B 0,C 180,E1 22458.5,E2 22458.5} C_VEL
LIN {X 0,Y 376.308,Z 1030.685,A -85,B 0,C 180,E1 22461.123,E2 22461.123} C_VEL
LIN {X 0,Y 381.328,Z 1011.447,A -85,B 0,C 180,E1 22462.164,E2 22462.164} C_VEL
LIN {X 0,Y 373.042,Z 984.965,A -85,B 0,C 180,E1 22466.585,E2 22466.585} C_VEL
LIN {X 0,Y 362.199,Z 960.262,A -85,B 0,C 180,E1 22471.806,E2 22471.806} C_VEL
LIN {X 0,Y 351.737,Z 941.884,A -85,B 0,C 180,E1 22477.197,E2 22477.197} C_VEL
LIN {X 0,Y 344.738,Z 930.775,A -85,B 0,C 180,E1 22481.675,E2 22481.675} C_VEL
LIN {X 0,Y 340.631,Z 924.729,A -85,B 0,C 180,E1 22485.023,E2 22485.023} C_VEL
LIN {X 0,Y 338.157,Z 920.374,A -85,B 0,C 180,E1 22487.718,E2 22487.718} C_VEL
LIN {X 0,Y 335.097,Z 913.991,A -85,B 0,C 180,E1 22493.513,E2 22493.513} C_VEL
LIN {X 0,Y 335.439,Z 914.649,A -85,B 0,C 180,E1 22501.54,E2 22501.54} C_VEL
LIN {X 0,Y 339.644,Z 922.546,A -85,B 0,C 180,E1 22508.009,E2 22508.009} C_VEL
LIN {X 0,Y 344.424,Z 930.489,A -85,B 0,C 180,E1 22512.304,E2 22512.304} C_VEL
LIN {X 0,Y 351.261,Z 941.924,A -85,B 0,C 180,E1 22516.928,E2 22516.928} C_VEL
LIN {X 0,Y 360.749,Z 960.639,A -85,B 0,C 180,E1 22522.356,E2 22522.356} C_VEL
LIN {X 0,Y 370.073,Z 983.931,A -85,B 0,C 180,E1 22527.424,E2 22527.424} C_VEL
LIN {X 0,Y 377.379,Z 1011.375,A -85,B 0,C 180,E1 22532.137,E2 22532.137} C_VEL
LIN {X 0,Y 377.824,Z 1016.389,A -85,B 0,C 180,E1 22532.823,E2 22532.823} C_VEL
LIN {X 0,Y 365.364,Z 1055.616,A -85,B 0,C 180,E1 22535.488,E2 22535.488} C_VEL
LIN {X 0,Y 350.384,Z 1093.369,A -85,B 0,C 180,E1 22539.128,E2 22539.128} C_VEL
LIN {X 0,Y 333.987,Z 1128.786,A -85,B 0,C 180,E1 22544.012,E2 22544.012} C_VEL
LIN {X 0,Y 318.24,Z 1159.449,A -85,B 0,C 180,E1 22550.026,E2 22550.026} C_VEL
LIN {X 0,Y 305.445,Z 1184.139,A -85,B 0,C 180,E1 22556.927,E2 22556.927} C_VEL
LIN {X 0,Y 295.682,Z 1204.122,A -85,B 0,C 180,E1 22564.991,E2 22564.991} C_VEL
LIN {X 0,Y 290.354,Z 1217.752,A -85,B 0,C 180,E1 22573.319,E2 22573.319} C_VEL
LIN {X 0,Y 288.525,Z 1225.316,A -85,B 0,C 180,E1 22580.935,E2 22580.935} C_VEL
LIN {X 0,Y 288.248,Z 1228.154,A -85,B 0,C 180,E1 22586.986,E2 22586.986} C_VEL
LIN {X 0,Y 288.248,Z 1228.158,A -85,B 0,C 180,E1 22593.013,E2 22593.013} C_VEL
LIN {X 0,Y 288.717,Z 1224.149,A -85,B 0,C 180,E1 22600.585,E2 22600.585} C_VEL
LIN {X 0,Y 291.392,Z 1214.709,A -85,B 0,C 180,E1 22608.966,E2 22608.966} C_VEL
LIN {X 0,Y 297.863,Z 1199.391,A -85,B 0,C 180,E1 22617.248,E2 22617.248} C_VEL
LIN {X 0,Y 308.828,Z 1177.492,A -85,B 0,C 180,E1 22625.206,E2 22625.206} C_VEL
LIN {X 0,Y 323.032,Z 1150.614,A -85,B 0,C 180,E1 22631.947,E2 22631.947} C_VEL
LIN {X 0,Y 338.08,Z 1120.596,A -85,B 0,C 180,E1 22637.292,E2 22637.292} C_VEL
LIN {X 0,Y 352.87,Z 1087.881,A -85,B 0,C 180,E1 22641.501,E2 22641.501} C_VEL
LIN {X 0,Y 367.763,Z 1049.323,A -85,B 0,C 180,E1 22645.025,E2 22645.025} C_VEL
LIN {X 0,Y 378.3,Z 1015.242,A -85,B 0,C 180,E1 22647.262,E2 22647.262} C_VEL
LIN {X 0,Y 371.703,Z 988.737,A -85,B 0,C 180,E1 22651.716,E2 22651.716} C_VEL
LIN {X 0,Y 362.772,Z 964.599,A -85,B 0,C 180,E1 22656.711,E2 22656.711} C_VEL
LIN {X 0,Y 352.233,Z 943.353,A -85,B 0,C 180,E1 22662.637,E2 22662.637} C_VEL
LIN {X 0,Y 344.677,Z 930.802,A -85,B 0,C 180,E1 22667.705,E2 22667.705} C_VEL
LIN {X 0,Y 341.477,Z 925.622,A -85,B 0,C 180,E1 22670.42,E2 22670.42} C_VEL
LIN {X 0,Y 338.332,Z 920.168,A -85,B 0,C 180,E1 22673.859,E2 22673.859} C_VEL
LIN {X 0,Y 336.048,Z 916.695,A -85,B 0,C 180,E1 22677.474,E2 22677.474} C_VEL
LIN {X 0,Y 335.008,Z 917.133,A -85,B 0,C 180,E1 22679.699,E2 22679.699} C_VEL
LIN {X 0,Y 333.943,Z 921.65,A -85,B 0,C 180,E1 22683.446,E2 22683.446} C_VEL
LIN {X 0,Y 334.398,Z 922.846,A -85,B 0,C 180,E1 22686.39,E2 22686.39} C_VEL
LIN {X 0,Y 338.505,Z 930.369,A -85,B 0,C 180,E1 22693.42,E2 22693.42} C_VEL
LIN {X 0,Y 345.22,Z 940.921,A -85,B 0,C 180,E1 22699.211,E2 22699.211} C_VEL
LIN {X 0,Y 355.731,Z 959.999,A -85,B 0,C 180,E1 22705.68,E2 22705.68} C_VEL
LIN {X 0,Y 365.479,Z 981.357,A -85,B 0,C 180,E1 22710.856,E2 22710.856} C_VEL
LIN {X 0,Y 374.041,Z 1006.394,A -85,B 0,C 180,E1 22715.535,E2 22715.535} C_VEL
LIN {X 0,Y 376.113,Z 1015.868,A -85,B 0,C 180,E1 22717.012,E2 22717.012} C_VEL
LIN {X 0,Y 363.664,Z 1054.679,A -85,B 0,C 180,E1 22719.336,E2 22719.336} C_VEL
LIN {X 0,Y 348.548,Z 1091.093,A -85,B 0,C 180,E1 22722.579,E2 22722.579} C_VEL
LIN {X 0,Y 331.919,Z 1124.157,A -85,B 0,C 180,E1 22726.902,E2 22726.902} C_VEL
LIN {X 0,Y 315.739,Z 1152.415,A -85,B 0,C 180,E1 22732.329,E2 22732.329} C_VEL
LIN {X 0,Y 300.657,Z 1176.664,A -85,B 0,C 180,E1 22739.236,E2 22739.236} C_VEL
LIN {X 0,Y 289.86,Z 1194.318,A -85,B 0,C 180,E1 22746.917,E2 22746.917} C_VEL
LIN {X 0,Y 283.747,Z 1205.433,A -85,B 0,C 180,E1 22754.514,E2 22754.514} C_VEL
LIN {X 0,Y 281.29,Z 1210.959,A -85,B 0,C 180,E1 22760.7,E2 22760.7} C_VEL
LIN {X 0,Y 280.5,Z 1213.66,A -85,B 0,C 180,E1 22766.904,E2 22766.904} C_VEL
LIN {X 0,Y 280.527,Z 1213.622,A -85,B 0,C 180,E1 22773.097,E2 22773.097} C_VEL
LIN {X 0,Y 281.841,Z 1209.707,A -85,B 0,C 180,E1 22780.847,E2 22780.847} C_VEL
LIN {X 0,Y 286.412,Z 1200.27,A -85,B 0,C 180,E1 22789.309,E2 22789.309} C_VEL
LIN {X 0,Y 294.483,Z 1186.474,A -85,B 0,C 180,E1 22796.76,E2 22796.76} C_VEL
LIN {X 0,Y 306.732,Z 1166.87,A -85,B 0,C 180,E1 22803.764,E2 22803.764} C_VEL
LIN {X 0,Y 321.117,Z 1143.11,A -85,B 0,C 180,E1 22809.572,E2 22809.572} C_VEL
LIN {X 0,Y 337.423,Z 1113.507,A -85,B 0,C 180,E1 22814.561,E2 22814.561} C_VEL
LIN {X 0,Y 353.718,Z 1079.046,A -85,B 0,C 180,E1 22818.529,E2 22818.529} C_VEL
LIN {X 0,Y 368.042,Z 1041.515,A -85,B 0,C 180,E1 22821.469,E2 22821.469} C_VEL
LIN {X 0,Y 375.982,Z 1014.59,A -85,B 0,C 180,E1 22823.001,E2 22823.001} C_VEL
LIN {X 0,Y 368.013,Z 988.015,A -85,B 0,C 180,E1 22827.651,E2 22827.651} C_VEL
LIN {X 0,Y 358.449,Z 965.741,A -85,B 0,C 180,E1 22832.608,E2 22832.608} C_VEL
LIN {X 0,Y 348.98,Z 947.901,A -85,B 0,C 180,E1 22837.986,E2 22837.986} C_VEL
LIN {X 0,Y 341.23,Z 934.77,A -85,B 0,C 180,E1 22843.563,E2 22843.563} C_VEL
LIN {X 0,Y 336.689,Z 927.776,A -85,B 0,C 180,E1 22848.322,E2 22848.322} C_VEL
LIN {X 0,Y 333.952,Z 921.755,A -85,B 0,C 180,E1 22854.145,E2 22854.145} C_VEL
LIN {X 0,Y 334.404,Z 922.492,A -85,B 0,C 180,E1 22861.383,E2 22861.383} C_VEL
LIN {X 0,Y 338.219,Z 930.153,A -85,B 0,C 180,E1 22867.726,E2 22867.726} C_VEL
LIN {X 0,Y 343.099,Z 938.592,A -85,B 0,C 180,E1 22872.272,E2 22872.272} C_VEL
LIN {X 0,Y 350.749,Z 952.436,A -85,B 0,C 180,E1 22877.682,E2 22877.682} C_VEL
LIN {X 0,Y 360.038,Z 973.282,A -85,B 0,C 180,E1 22883.374,E2 22883.374} C_VEL
LIN {X 0,Y 367.548,Z 995.444,A -85,B 0,C 180,E1 22887.962,E2 22887.962} C_VEL
LIN {X 0,Y 372.539,Z 1019.031,A -85,B 0,C 180,E1 22891.976,E2 22891.976} C_VEL
LIN {X 0,Y 359.761,Z 1057.659,A -85,B 0,C 180,E1 22894.655,E2 22894.655} C_VEL
LIN {X 0,Y 344.767,Z 1094.149,A -85,B 0,C 180,E1 22898.221,E2 22898.221} C_VEL
LIN {X 0,Y 328.675,Z 1127.972,A -85,B 0,C 180,E1 22902.91,E2 22902.91} C_VEL
LIN {X 0,Y 312.246,Z 1158.766,A -85,B 0,C 180,E1 22908.957,E2 22908.957} C_VEL
LIN {X 0,Y 298.59,Z 1183.889,A -85,B 0,C 180,E1 22916.066,E2 22916.066} C_VEL
LIN {X 0,Y 288.159,Z 1204.233,A -85,B 0,C 180,E1 22924.468,E2 22924.468} C_VEL
LIN {X 0,Y 282.622,Z 1217.539,A -85,B 0,C 180,E1 22932.849,E2 22932.849} C_VEL
LIN {X 0,Y 280.646,Z 1225.111,A -85,B 0,C 180,E1 22940.678,E2 22940.678} C_VEL
LIN {X 0,Y 280.337,Z 1227.952,A -85,B 0,C 180,E1 22946.901,E2 22946.901} C_VEL
LIN {X 0,Y 280.337,Z 1227.956,A -85,B 0,C 180,E1 22953.098,E2 22953.098} C_VEL
LIN {X 0,Y 280.852,Z 1223.942,A -85,B 0,C 180,E1 22960.885,E2 22960.885} C_VEL
LIN {X 0,Y 283.737,Z 1214.552,A -85,B 0,C 180,E1 22969.458,E2 22969.458} C_VEL
LIN {X 0,Y 290.588,Z 1199.166,A -85,B 0,C 180,E1 22977.989,E2 22977.989} C_VEL
LIN {X 0,Y 302.149,Z 1177.246,A -85,B 0,C 180,E1 22986.105,E2 22986.105} C_VEL
LIN {X 0,Y 317.016,Z 1150.339,A -85,B 0,C 180,E1 22992.932,E2 22992.932} C_VEL
LIN {X 0,Y 332.917,Z 1119.586,A -85,B 0,C 180,E1 22998.432,E2 22998.432} C_VEL
LIN {X 0,Y 348.783,Z 1085.336,A -85,B 0,C 180,E1 23002.775,E2 23002.775} C_VEL
LIN {X 0,Y 363.177,Z 1048.737,A -85,B 0,C 180,E1 23006.073,E2 23006.073} C_VEL
LIN {X 0,Y 372.864,Z 1018.152,A -85,B 0,C 180,E1 23008.114,E2 23008.114} C_VEL
LIN {X 0,Y 367.274,Z 993.877,A -85,B 0,C 180,E1 23012.349,E2 23012.349} C_VEL
LIN {X 0,Y 358.921,Z 970.122,A -85,B 0,C 180,E1 23017.431,E2 23017.431} C_VEL
LIN {X 0,Y 349.558,Z 949.928,A -85,B 0,C 180,E1 23023.23,E2 23023.23} C_VEL
LIN {X 0,Y 341.973,Z 936.3,A -85,B 0,C 180,E1 23028.902,E2 23028.902} C_VEL
LIN {X 0,Y 336.975,Z 927.782,A -85,B 0,C 180,E1 23034.211,E2 23034.211} C_VEL
LIN {X 0,Y 334.359,Z 921.662,A -85,B 0,C 180,E1 23039.996,E2 23039.996} C_VEL
LIN {X 0,Y 333.943,Z 921.65,A -85,B 0,C 180,E1 23043.446,E2 23043.446} C_VEL
LIN {X 0,Y 333.896,Z 925.036,A -85,B 0,C 180,E1 23045.615,E2 23045.615} C_VEL
LIN {X 0,Y 334.259,Z 933.902,A -85,B 0,C 180,E1 23049.121,E2 23049.121} C_VEL
LIN {X 0,Y 337.092,Z 938.01,A -85,B 0,C 180,E1 23053.147,E2 23053.147} C_VEL
LIN {X 0,Y 343.308,Z 948.392,A -85,B 0,C 180,E1 23058.865,E2 23058.865} C_VEL
LIN {X 0,Y 352.718,Z 966.543,A -85,B 0,C 180,E1 23065.156,E2 23065.156} C_VEL
LIN {X 0,Y 361.873,Z 987.882,A -85,B 0,C 180,E1 23070.412,E2 23070.412} C_VEL
LIN {X 0,Y 369.403,Z 1011.912,A -85,B 0,C 180,E1 23075.035,E2 23075.035} C_VEL
LIN {X 0,Y 370.855,Z 1018.793,A -85,B 0,C 180,E1 23076.144,E2 23076.144} C_VEL
LIN {X 0,Y 357.506,Z 1058.464,A -85,B 0,C 180,E1 23078.605,E2 23078.605} C_VEL
LIN {X 0,Y 342.106,Z 1093.912,A -85,B 0,C 180,E1 23081.869,E2 23081.869} C_VEL
LIN {X 0,Y 325.233,Z 1126.14,A -85,B 0,C 180,E1 23086.218,E2 23086.218} C_VEL
LIN {X 0,Y 308.597,Z 1154.052,A -85,B 0,C 180,E1 23091.755,E2 23091.755} C_VEL
LIN {X 0,Y 294.044,Z 1176.498,A -85,B 0,C 180,E1 23098.288,E2 23098.288} C_VEL
LIN {X 0,Y 282.296,Z 1194.843,A -85,B 0,C 180,E1 23106.466,E2 23106.466} C_VEL
LIN {X 0,Y 276.074,Z 1205.639,A -85,B 0,C 180,E1 23114.072,E2 23114.072} C_VEL
LIN {X 0,Y 273.456,Z 1211.163,A -85,B 0,C 180,E1 23120.431,E2 23120.431} C_VEL
LIN {X 0,Y 272.62,Z 1213.862,A -85,B 0,C 180,E1 23126.814,E2 23126.814} C_VEL
LIN {X 0,Y 272.636,Z 1213.824,A -85,B 0,C 180,E1 23133.187,E2 23133.187} C_VEL
LIN {X 0,Y 274.041,Z 1209.913,A -85,B 0,C 180,E1 23141.159,E2 23141.159} C_VEL
LIN {X 0,Y 278.894,Z 1200.479,A -85,B 0,C 180,E1 23149.851,E2 23149.851} C_VEL
LIN {X 0,Y 288.422,Z 1185.015,A -85,B 0,C 180,E1 23158.219,E2 23158.219} C_VEL
LIN {X 0,Y 301.579,Z 1164.773,A -85,B 0,C 180,E1 23165.298,E2 23165.298} C_VEL
LIN {X 0,Y 316.852,Z 1140.26,A -85,B 0,C 180,E1 23171.115,E2 23171.115} C_VEL
LIN {X 0,Y 332.904,Z 1111.774,A -85,B 0,C 180,E1 23175.8,E2 23175.8} C_VEL
LIN {X 0,Y 349.045,Z 1078.348,A -85,B 0,C 180,E1 23179.605,E2 23179.605} C_VEL
LIN {X 0,Y 363.189,Z 1042.165,A -85,B 0,C 180,E1 23182.441,E2 23182.441} C_VEL
LIN {X 0,Y 370.706,Z 1017.79,A -85,B 0,C 180,E1 23183.857,E2 23183.857} C_VEL
LIN {X 0,Y 363.275,Z 991.914,A -85,B 0,C 180,E1 23188.587,E2 23188.587} C_VEL
LIN {X 0,Y 354.333,Z 970.172,A -85,B 0,C 180,E1 23193.671,E2 23193.671} C_VEL
LIN {X 0,Y 345.469,Z 952.772,A -85,B 0,C 180,E1 23199.23,E2 23199.23} C_VEL
LIN {X 0,Y 338.735,Z 941.255,A -85,B 0,C 180,E1 23204.688,E2 23204.688} C_VEL
LIN {X 0,Y 335.457,Z 935.53,A -85,B 0,C 180,E1 23208.444,E2 23208.444} C_VEL
LIN {X 0,Y 332.786,Z 929.511,A -85,B 0,C 180,E1 23214.78,E2 23214.78} C_VEL
LIN {X 0,Y 333.268,Z 930.289,A -85,B 0,C 180,E1 23221.224,E2 23221.224} C_VEL
LIN {X 0,Y 336.756,Z 937.773,A -85,B 0,C 180,E1 23227.435,E2 23227.435} C_VEL
LIN {X 0,Y 341.084,Z 945.973,A -85,B 0,C 180,E1 23231.939,E2 23231.939} C_VEL
LIN {X 0,Y 347.899,Z 959.128,A -85,B 0,C 180,E1 23237.178,E2 23237.178} C_VEL
LIN {X 0,Y 356.528,Z 979.705,A -85,B 0,C 180,E1 23242.899,E2 23242.899} C_VEL
LIN {X 0,Y 363.345,Z 1002.099,A -85,B 0,C 180,E1 23247.639,E2 23247.639} C_VEL
LIN {X 0,Y 367.255,Z 1021.972,A -85,B 0,C 180,E1 23251.123,E2 23251.123} C_VEL
LIN {X 0,Y 353.83,Z 1060.7,A -85,B 0,C 180,E1 23253.874,E2 23253.874} C_VEL
LIN {X 0,Y 338.146,Z 1097.286,A -85,B 0,C 180,E1 23257.569,E2 23257.569} C_VEL
LIN {X 0,Y 322.095,Z 1129.619,A -85,B 0,C 180,E1 23262.186,E2 23262.186} C_VEL
LIN {X 0,Y 305.686,Z 1159.219,A -85,B 0,C 180,E1 23268.129,E2 23268.129} C_VEL
LIN {X 0,Y 291.794,Z 1183.639,A -85,B 0,C 180,E1 23275.163,E2 23275.163} C_VEL
LIN {X 0,Y 280.759,Z 1204.118,A -85,B 0,C 180,E1 23283.806,E2 23283.806} C_VEL
LIN {X 0,Y 274.927,Z 1217.325,A -85,B 0,C 180,E1 23292.353,E2 23292.353} C_VEL
LIN {X 0,Y 272.769,Z 1224.906,A -85,B 0,C 180,E1 23300.406,E2 23300.406} C_VEL
LIN {X 0,Y 272.437,Z 1227.75,A -85,B 0,C 180,E1 23306.811,E2 23306.811} C_VEL
LIN {X 0,Y 272.437,Z 1227.754,A -85,B 0,C 180,E1 23313.188,E2 23313.188} C_VEL
LIN {X 0,Y 273.02,Z 1223.737,A -85,B 0,C 180,E1 23321.201,E2 23321.201} C_VEL
LIN {X 0,Y 275.683,Z 1215.347,A -85,B 0,C 180,E1 23329.256,E2 23329.256} C_VEL
LIN {X 0,Y 282.442,Z 1200.777,A -85,B 0,C 180,E1 23337.869,E2 23337.869} C_VEL
LIN {X 0,Y 292.99,Z 1181.497,A -85,B 0,C 180,E1 23345.579,E2 23345.579} C_VEL
LIN {X 0,Y 307.432,Z 1156.275,A -85,B 0,C 180,E1 23352.596,E2 23352.596} C_VEL
LIN {X 0,Y 324.607,Z 1125.036,A -85,B 0,C 180,E1 23358.604,E2 23358.604} C_VEL
LIN {X 0,Y 341.544,Z 1090.405,A -85,B 0,C 180,E1 23363.258,E2 23363.258} C_VEL
LIN {X 0,Y 357.863,Z 1050.628,A -85,B 0,C 180,E1 23366.96,E2 23366.96} C_VEL
LIN {X 0,Y 367.503,Z 1020.895,A -85,B 0,C 180,E1 23369.015,E2 23369.015} C_VEL
LIN {X 0,Y 361.96,Z 995.966,A -85,B 0,C 180,E1 23373.593,E2 23373.593} C_VEL
LIN {X 0,Y 353.938,Z 972.672,A -85,B 0,C 180,E1 23378.909,E2 23378.909} C_VEL
LIN {X 0,Y 345.391,Z 953.38,A -85,B 0,C 180,E1 23384.902,E2 23384.902} C_VEL
LIN {X 0,Y 338.521,Z 941.013,A -85,B 0,C 180,E1 23390.823,E2 23390.823} C_VEL
LIN {X 0,Y 335.582,Z 935.418,A -85,B 0,C 180,E1 23394.502,E2 23394.502} C_VEL
LIN {X 0,Y 333.316,Z 929.48,A -85,B 0,C 180,E1 23399.996,E2 23399.996} C_VEL
LIN {X 0,Y 333.292,Z 930.497,A -85,B 0,C 180,E1 23406.112,E2 23406.112} C_VEL
LIN {X 0,Y 334.259,Z 933.902,A -85,B 0,C 180,E1 23409.121,E2 23409.121} C_VEL
LIN {X 0,Y 334.801,Z 939.209,A -85,B 0,C 180,E1 23410.916,E2 23410.916} C_VEL
LIN {X 0,Y 335.441,Z 945.238,A -85,B 0,C 180,E1 23412.677,E2 23412.677} C_VEL
LIN {X 0,Y 341.342,Z 955.984,A -85,B 0,C 180,E1 23418.592,E2 23418.592} C_VEL
LIN {X 0,Y 350.111,Z 973.919,A -85,B 0,C 180,E1 23424.871,E2 23424.871} C_VEL
LIN {X 0,Y 357.884,Z 993.575,A -85,B 0,C 180,E1 23429.822,E2 23429.822} C_VEL
LIN {X 0,Y 365.042,Z 1018.51,A -85,B 0,C 180,E1 23434.718,E2 23434.718} C_VEL
LIN {X 0,Y 365.626,Z 1021.599,A -85,B 0,C 180,E1 23435.257,E2 23435.257} C_VEL
LIN {X 0,Y 352.644,Z 1058.958,A -85,B 0,C 180,E1 23437.604,E2 23437.604} C_VEL
LIN {X 0,Y 336.87,Z 1094.276,A -85,B 0,C 180,E1 23440.866,E2 23440.866} C_VEL
LIN {X 0,Y 319.246,Z 1126.915,A -85,B 0,C 180,E1 23445.314,E2 23445.314} C_VEL
LIN {X 0,Y 302.356,Z 1154.3,A -85,B 0,C 180,E1 23450.816,E2 23450.816} C_VEL
LIN {X 0,Y 286.896,Z 1177.242,A -85,B 0,C 180,E1 23457.647,E2 23457.647} C_VEL
LIN {X 0,Y 275.494,Z 1194.3,A -85,B 0,C 180,E1 23465.346,E2 23465.346} C_VEL
LIN {X 0,Y 268.424,Z 1205.846,A -85,B 0,C 180,E1 23473.605,E2 23473.605} C_VEL
LIN {X 0,Y 265.621,Z 1211.368,A -85,B 0,C 180,E1 23480.146,E2 23480.146} C_VEL
LIN {X 0,Y 264.718,Z 1214.064,A -85,B 0,C 180,E1 23486.719,E2 23486.719} C_VEL
LIN {X 0,Y 264.735,Z 1214.027,A -85,B 0,C 180,E1 23493.282,E2 23493.282} C_VEL
LIN {X 0,Y 266.248,Z 1210.116,A -85,B 0,C 180,E1 23501.49,E2 23501.49} C_VEL
LIN {X 0,Y 271.383,Z 1200.688,A -85,B 0,C 180,E1 23510.425,E2 23510.425} C_VEL
LIN {X 0,Y 280.265,Z 1186.921,A -85,B 0,C 180,E1 23518.235,E2 23518.235} C_VEL
LIN {X 0,Y 293.546,Z 1167.362,A -85,B 0,C 180,E1 23525.502,E2 23525.502} C_VEL
LIN {X 0,Y 308.992,Z 1143.675,A -85,B 0,C 180,E1 23531.456,E2 23531.456} C_VEL
LIN {X 0,Y 326.882,Z 1113.154,A -85,B 0,C 180,E1 23536.653,E2 23536.653} C_VEL
LIN {X 0,Y 343.566,Z 1079.75,A -85,B 0,C 180,E1 23540.52,E2 23540.52} C_VEL
LIN {X 0,Y 358.451,Z 1042.814,A -85,B 0,C 180,E1 23543.437,E2 23543.437} C_VEL
LIN {X 0,Y 365.358,Z 1020.988,A -85,B 0,C 180,E1 23544.729,E2 23544.729} C_VEL
LIN {X 0,Y 358.544,Z 995.824,A -85,B 0,C 180,E1 23549.539,E2 23549.539} C_VEL
LIN {X 0,Y 350.338,Z 974.577,A -85,B 0,C 180,E1 23554.76,E2 23554.76} C_VEL
LIN {X 0,Y 342.224,Z 958.195,A -85,B 0,C 180,E1 23560.382,E2 23560.382} C_VEL
LIN {X 0,Y 336.73,Z 948.368,A -85,B 0,C 180,E1 23565.262,E2 23565.262} C_VEL
LIN {X 0,Y 333.97,Z 943.012,A -85,B 0,C 180,E1 23568.889,E2 23568.889} C_VEL
LIN {X 0,Y 331.652,Z 937.321,A -85,B 0,C 180,E1 23574.762,E2 23574.762} C_VEL
LIN {X 0,Y 332.048,Z 938.122,A -85,B 0,C 180,E1 23581.066,E2 23581.066} C_VEL
LIN {X 0,Y 335.087,Z 945.465,A -85,B 0,C 180,E1 23587.227,E2 23587.227} C_VEL
LIN {X 0,Y 340.388,Z 955.557,A -85,B 0,C 180,E1 23592.779,E2 23592.779} C_VEL
LIN {X 0,Y 347.643,Z 972.249,A -85,B 0,C 180,E1 23598.667,E2 23598.667} C_VEL
LIN {X 0,Y 354.931,Z 992.373,A -85,B 0,C 180,E1 23603.924,E2 23603.924} C_VEL
LIN {X 0,Y 360.676,Z 1016.304,A -85,B 0,C 180,E1 23608.748,E2 23608.748} C_VEL
LIN {X 0,Y 361.671,Z 1025.979,A -85,B 0,C 180,E1 23610.312,E2 23610.312} C_VEL
LIN {X 0,Y 347.264,Z 1065.641,A -85,B 0,C 180,E1 23613.237,E2 23613.237} C_VEL
LIN {X 0,Y 330.136,Z 1103.455,A -85,B 0,C 180,E1 23617.264,E2 23617.264} C_VEL
LIN {X 0,Y 311.646,Z 1138.252,A -85,B 0,C 180,E1 23622.658,E2 23622.658} C_VEL
LIN {X 0,Y 294.267,Z 1168.049,A -85,B 0,C 180,E1 23629.45,E2 23629.45} C_VEL
LIN {X 0,Y 280.368,Z 1191.499,A -85,B 0,C 180,E1 23637.284,E2 23637.284} C_VEL
LIN {X 0,Y 270.727,Z 1209.117,A -85,B 0,C 180,E1 23646.059,E2 23646.059} C_VEL
LIN {X 0,Y 266.148,Z 1220.229,A -85,B 0,C 180,E1 23654.702,E2 23654.702} C_VEL
LIN {X 0,Y 264.555,Z 1226.474,A -85,B 0,C 180,E1 23663.422,E2 23663.422} C_VEL
LIN {X 0,Y 264.734,Z 1227.913,A -85,B 0,C 180,E1 23670,E2 23670} C_VEL
LIN {X 0,Y 264.556,Z 1226.486,A -85,B 0,C 180,E1 23676.577,E2 23676.577} C_VEL
LIN {X 0,Y 266.118,Z 1220.387,A -85,B 0,C 180,E1 23685.178,E2 23685.178} C_VEL
LIN {X 0,Y 270.723,Z 1209.184,A -85,B 0,C 180,E1 23693.941,E2 23693.941} C_VEL
LIN {X 0,Y 280.362,Z 1191.583,A -85,B 0,C 180,E1 23702.716,E2 23702.716} C_VEL
LIN {X 0,Y 295.047,Z 1166.907,A -85,B 0,C 180,E1 23710.905,E2 23710.905} C_VEL
LIN {X 0,Y 312.658,Z 1136.688,A -85,B 0,C 180,E1 23717.653,E2 23717.653} C_VEL
LIN {X 0,Y 330.735,Z 1102.572,A -85,B 0,C 180,E1 23722.864,E2 23722.864} C_VEL
LIN {X 0,Y 347.819,Z 1064.697,A -85,B 0,C 180,E1 23726.864,E2 23726.864} C_VEL
LIN {X 0,Y 362.241,Z 1024.145,A -85,B 0,C 180,E1 23729.874,E2 23729.874} C_VEL
LIN {X 0,Y 357.067,Z 999.39,A -85,B 0,C 180,E1 23734.592,E2 23734.592} C_VEL
LIN {X 0,Y 349.96,Z 977.682,A -85,B 0,C 180,E1 23739.818,E2 23739.818} C_VEL
LIN {X 0,Y 342.455,Z 959.855,A -85,B 0,C 180,E1 23745.588,E2 23745.588} C_VEL
LIN {X 0,Y 336.546,Z 948.283,A -85,B 0,C 180,E1 23751.258,E2 23751.258} C_VEL
LIN {X 0,Y 333.941,Z 942.892,A -85,B 0,C 180,E1 23754.954,E2 23754.954} C_VEL
LIN {X 0,Y 332.167,Z 937.314,A -85,B 0,C 180,E1 23759.996,E2 23759.996} C_VEL
LIN {X 0,Y 332.106,Z 938.304,A -85,B 0,C 180,E1 23765.969,E2 23765.969} C_VEL
LIN {X 0,Y 335.441,Z 945.238,A -85,B 0,C 180,E1 23772.677,E2 23772.677} C_VEL
LIN {X 0,Y 336.709,Z 954.235,A -85,B 0,C 180,E1 23775.267,E2 23775.267} C_VEL
LIN {X 0,Y 338.488,Z 962.167,A -85,B 0,C 180,E1 23777.693,E2 23777.693} C_VEL
LIN {X 0,Y 338.701,Z 962.436,A -85,B 0,C 180,E1 23777.868,E2 23777.868} C_VEL
LIN {X 0,Y 346.643,Z 979.883,A -85,B 0,C 180,E1 23784.192,E2 23784.192} C_VEL
LIN {X 0,Y 354.234,Z 1000.426,A -85,B 0,C 180,E1 23789.487,E2 23789.487} C_VEL
LIN {X 0,Y 360.137,Z 1023.405,A -85,B 0,C 180,E1 23794.123,E2 23794.123} C_VEL
LIN {X 0,Y 359.286,Z 1028.2,A -85,B 0,C 180,E1 23794.542,E2 23794.542} C_VEL
LIN {X 0,Y 345.304,Z 1065.54,A -85,B 0,C 180,E1 23797.05,E2 23797.05} C_VEL
LIN {X 0,Y 329.342,Z 1099.251,A -85,B 0,C 180,E1 23800.372,E2 23800.372} C_VEL
LIN {X 0,Y 312.094,Z 1129.737,A -85,B 0,C 180,E1 23804.732,E2 23804.732} C_VEL
LIN {X 0,Y 295.327,Z 1155.805,A -85,B 0,C 180,E1 23810.162,E2 23810.162} C_VEL
LIN {X 0,Y 280.179,Z 1177.465,A -85,B 0,C 180,E1 23816.773,E2 23816.773} C_VEL
LIN {X 0,Y 268.266,Z 1194.478,A -85,B 0,C 180,E1 23824.614,E2 23824.614} C_VEL
LIN {X 0,Y 260.767,Z 1206.054,A -85,B 0,C 180,E1 23833.11,E2 23833.11} C_VEL
LIN {X 0,Y 257.792,Z 1211.572,A -85,B 0,C 180,E1 23839.844,E2 23839.844} C_VEL
LIN {X 0,Y 256.817,Z 1214.266,A -85,B 0,C 180,E1 23846.618,E2 23846.618} C_VEL
LIN {X 0,Y 256.834,Z 1214.23,A -85,B 0,C 180,E1 23853.383,E2 23853.383} C_VEL
LIN {X 0,Y 258.446,Z 1210.32,A -85,B 0,C 180,E1 23861.842,E2 23861.842} C_VEL
LIN {X 0,Y 263.897,Z 1200.9,A -85,B 0,C 180,E1 23871.032,E2 23871.032} C_VEL
LIN {X 0,Y 273.238,Z 1187.145,A -85,B 0,C 180,E1 23879.029,E2 23879.029} C_VEL
LIN {X 0,Y 287.061,Z 1167.604,A -85,B 0,C 180,E1 23886.431,E2 23886.431} C_VEL
LIN {X 0,Y 304.032,Z 1142.388,A -85,B 0,C 180,E1 23892.771,E2 23892.771} C_VEL
LIN {X 0,Y 321.507,Z 1113.498,A -85,B 0,C 180,E1 23897.678,E2 23897.678} C_VEL
LIN {X 0,Y 338.587,Z 1080.216,A -85,B 0,C 180,E1 23901.552,E2 23901.552} C_VEL
LIN {X 0,Y 354.287,Z 1042.117,A -85,B 0,C 180,E1 23904.542,E2 23904.542} C_VEL
LIN {X 0,Y 360.038,Z 1025.354,A -85,B 0,C 180,E1 23905.483,E2 23905.483} C_VEL
LIN {X 0,Y 355.674,Z 1005.47,A -85,B 0,C 180,E1 23909.266,E2 23909.266} C_VEL
LIN {X 0,Y 348.25,Z 984.042,A -85,B 0,C 180,E1 23914.435,E2 23914.435} C_VEL
LIN {X 0,Y 340.725,Z 967.061,A -85,B 0,C 180,E1 23920.025,E2 23920.025} C_VEL
LIN {X 0,Y 334.948,Z 955.897,A -85,B 0,C 180,E1 23925.52,E2 23925.52} C_VEL
LIN {X 0,Y 332.166,Z 950.474,A -85,B 0,C 180,E1 23929.326,E2 23929.326} C_VEL
LIN {X 0,Y 330.363,Z 945.104,A -85,B 0,C 180,E1 23934.742,E2 23934.742} C_VEL
LIN {X 0,Y 330.586,Z 945.769,A -85,B 0,C 180,E1 23940.824,E2 23940.824} C_VEL
LIN {X 0,Y 333.424,Z 953.241,A -85,B 0,C 180,E1 23947.099,E2 23947.099} C_VEL
LIN {X 0,Y 338.103,Z 963.112,A -85,B 0,C 180,E1 23952.538,E2 23952.538} C_VEL
LIN {X 0,Y 344.671,Z 979.315,A -85,B 0,C 180,E1 23958.336,E2 23958.336} C_VEL
LIN {X 0,Y 351.297,Z 999.657,A -85,B 0,C 180,E1 23963.702,E2 23963.702} C_VEL
LIN {X 0,Y 356.345,Z 1024.416,A -85,B 0,C 180,E1 23968.715,E2 23968.715} C_VEL
LIN {X 0,Y 356.512,Z 1028.673,A -85,B 0,C 180,E1 23969.407,E2 23969.407} C_VEL
LIN {X 0,Y 341.901,Z 1067.419,A -85,B 0,C 180,E1 23972.308,E2 23972.308} C_VEL
LIN {X 0,Y 324.014,Z 1105.486,A -85,B 0,C 180,E1 23976.44,E2 23976.44} C_VEL
LIN {X 0,Y 306.172,Z 1137.955,A -85,B 0,C 180,E1 23981.534,E2 23981.534} C_VEL
LIN {X 0,Y 288.081,Z 1167.794,A -85,B 0,C 180,E1 23988.389,E2 23988.389} C_VEL
LIN {X 0,Y 273.525,Z 1191.266,A -85,B 0,C 180,E1 23996.359,E2 23996.359} C_VEL
LIN {X 0,Y 263.337,Z 1208.896,A -85,B 0,C 180,E1 24005.343,E2 24005.343} C_VEL
LIN {X 0,Y 258.078,Z 1220.943,A -85,B 0,C 180,E1 24015.189,E2 24015.189} C_VEL
LIN {X 0,Y 256.683,Z 1226.271,A -85,B 0,C 180,E1 24023.219,E2 24023.219} C_VEL
LIN {X 0,Y 256.848,Z 1227.712,A -85,B 0,C 180,E1 24030,E2 24030} C_VEL
LIN {X 0,Y 256.683,Z 1226.284,A -85,B 0,C 180,E1 24036.78,E2 24036.78} C_VEL
LIN {X 0,Y 258.433,Z 1219.917,A -85,B 0,C 180,E1 24045.917,E2 24045.917} C_VEL
LIN {X 0,Y 263.33,Z 1208.966,A -85,B 0,C 180,E1 24054.657,E2 24054.657} C_VEL
LIN {X 0,Y 274.037,Z 1190.52,A -85,B 0,C 180,E1 24063.975,E2 24063.975} C_VEL
LIN {X 0,Y 288.876,Z 1166.641,A -85,B 0,C 180,E1 24071.974,E2 24071.974} C_VEL
LIN {X 0,Y 306.216,Z 1138.145,A -85,B 0,C 180,E1 24078.456,E2 24078.456} C_VEL
LIN {X 0,Y 325.036,Z 1103.911,A -85,B 0,C 180,E1 24083.792,E2 24083.792} C_VEL
LIN {X 0,Y 342.844,Z 1065.731,A -85,B 0,C 180,E1 24087.863,E2 24087.863} C_VEL
LIN {X 0,Y 356.903,Z 1026.871,A -85,B 0,C 180,E1 24090.836,E2 24090.836} C_VEL
LIN {X 0,Y 352.222,Z 1002.878,A -85,B 0,C 180,E1 24095.628,E2 24095.628} C_VEL
LIN {X 0,Y 345.986,Z 982.336,A -85,B 0,C 180,E1 24100.826,E2 24100.826} C_VEL
LIN {X 0,Y 339.579,Z 966.306,A -85,B 0,C 180,E1 24106.287,E2 24106.287} C_VEL
LIN {X 0,Y 334.523,Z 955.568,A -85,B 0,C 180,E1 24111.697,E2 24111.697} C_VEL
LIN {X 0,Y 332.23,Z 950.443,A -85,B 0,C 180,E1 24115.256,E2 24115.256} C_VEL
LIN {X 0,Y 330.664,Z 945.066,A -85,B 0,C 180,E1 24120.653,E2 24120.653} C_VEL
LIN {X 0,Y 330.734,Z 946.201,A -85,B 0,C 180,E1 24125.912,E2 24125.912} C_VEL
LIN {X 0,Y 333.888,Z 953.344,A -85,B 0,C 180,E1 24132.692,E2 24132.692} C_VEL
LIN {X 0,Y 338.701,Z 962.436,A -85,B 0,C 180,E1 24137.868,E2 24137.868} C_VEL
LIN {X 0,Y 340.205,Z 967.487,A -85,B 0,C 180,E1 24139.464,E2 24139.464} C_VEL
LIN {X 0,Y 341.866,Z 982.625,A -85,B 0,C 180,E1 24142.465,E2 24142.465} C_VEL
LIN {X 0,Y 342.074,Z 983.117,A -85,B 0,C 180,E1 24142.629,E2 24142.629} C_VEL
LIN {X 0,Y 349.251,Z 1003.011,A -85,B 0,C 180,E1 24148.169,E2 24148.169} C_VEL
LIN {X 0,Y 354.803,Z 1025.879,A -85,B 0,C 180,E1 24153.052,E2 24153.052} C_VEL
LIN {X 0,Y 354.377,Z 1030.638,A -85,B 0,C 180,E1 24153.596,E2 24153.596} C_VEL
LIN {X 0,Y 338.7,Z 1070.467,A -85,B 0,C 180,E1 24156.362,E2 24156.362} C_VEL
LIN {X 0,Y 320.876,Z 1105.921,A -85,B 0,C 180,E1 24160.079,E2 24160.079} C_VEL
LIN {X 0,Y 302.28,Z 1136.777,A -85,B 0,C 180,E1 24164.895,E2 24164.895} C_VEL
LIN {X 0,Y 283.924,Z 1163.51,A -85,B 0,C 180,E1 24171.164,E2 24171.164} C_VEL
LIN {X 0,Y 268.56,Z 1184.473,A -85,B 0,C 180,E1 24178.665,E2 24178.665} C_VEL
LIN {X 0,Y 257.162,Z 1200.18,A -85,B 0,C 180,E1 24187.481,E2 24187.481} C_VEL
LIN {X 0,Y 251.311,Z 1209.38,A -85,B 0,C 180,E1 24196.044,E2 24196.044} C_VEL
LIN {X 0,Y 249.221,Z 1213.468,A -85,B 0,C 180,E1 24203.016,E2 24203.016} C_VEL
LIN {X 0,Y 248.982,Z 1214.785,A -85,B 0,C 180,E1 24210,E2 24210} C_VEL
LIN {X 0,Y 249.243,Z 1213.402,A -85,B 0,C 180,E1 24216.984,E2 24216.984} C_VEL
LIN {X 0,Y 252.55,Z 1207.205,A -85,B 0,C 180,E1 24226.33,E2 24226.33} C_VEL
LIN {X 0,Y 261.26,Z 1194.307,A -85,B 0,C 180,E1 24236.224,E2 24236.224} C_VEL
LIN {X 0,Y 275.115,Z 1175.422,A -85,B 0,C 180,E1 24244.851,E2 24244.851} C_VEL
LIN {X 0,Y 292.128,Z 1151.729,A -85,B 0,C 180,E1 24251.794,E2 24251.794} C_VEL
LIN {X 0,Y 309.949,Z 1124.34,A -85,B 0,C 180,E1 24257.166,E2 24257.166} C_VEL
LIN {X 0,Y 328.153,Z 1091.881,A -85,B 0,C 180,E1 24261.471,E2 24261.471} C_VEL
LIN {X 0,Y 344.722,Z 1055.915,A -85,B 0,C 180,E1 24264.682,E2 24264.682} C_VEL
LIN {X 0,Y 354.985,Z 1027.603,A -85,B 0,C 180,E1 24266.495,E2 24266.495} C_VEL
LIN {X 0,Y 349.333,Z 1003.739,A -85,B 0,C 180,E1 24271.513,E2 24271.513} C_VEL
LIN {X 0,Y 342.155,Z 983.507,A -85,B 0,C 180,E1 24277.051,E2 24277.051} C_VEL
LIN {X 0,Y 335.639,Z 968.795,A -85,B 0,C 180,E1 24282.793,E2 24282.793} C_VEL
LIN {X 0,Y 330.938,Z 958.625,A -85,B 0,C 180,E1 24288.853,E2 24288.853} C_VEL
LIN {X 0,Y 328.877,Z 952.861,A -85,B 0,C 180,E1 24294.718,E2 24294.718} C_VEL
LIN {X 0,Y 329.033,Z 953.493,A -85,B 0,C 180,E1 24300.663,E2 24300.663} C_VEL
LIN {X 0,Y 331.419,Z 960.818,A -85,B 0,C 180,E1 24306.895,E2 24306.895} C_VEL
LIN {X 0,Y 335.729,Z 970.617,A -85,B 0,C 180,E1 24312.297,E2 24312.297} C_VEL
LIN {X 0,Y 341.266,Z 985.638,A -85,B 0,C 180,E1 24317.773,E2 24317.773} C_VEL
LIN {X 0,Y 347.127,Z 1005.373,A -85,B 0,C 180,E1 24323.13,E2 24323.13} C_VEL
LIN {X 0,Y 351.266,Z 1028.534,A -85,B 0,C 180,E1 24327.973,E2 24327.973} C_VEL
LIN {X 0,Y 350.994,Z 1032.628,A -85,B 0,C 180,E1 24328.551,E2 24328.551} C_VEL
LIN {X 0,Y 336.277,Z 1069.953,A -85,B 0,C 180,E1 24331.423,E2 24331.423} C_VEL
LIN {X 0,Y 318.976,Z 1105.621,A -85,B 0,C 180,E1 24335.332,E2 24335.332} C_VEL
LIN {X 0,Y 299.787,Z 1139.308,A -85,B 0,C 180,E1 24340.695,E2 24340.695} C_VEL
LIN {X 0,Y 281.99,Z 1167.541,A -85,B 0,C 180,E1 24347.28,E2 24347.28} C_VEL
LIN {X 0,Y 266.79,Z 1191.033,A -85,B 0,C 180,E1 24355.391,E2 24355.391} C_VEL
LIN {X 0,Y 255.971,Z 1208.675,A -85,B 0,C 180,E1 24364.584,E2 24364.584} C_VEL
LIN {X 0,Y 250.461,Z 1220.253,A -85,B 0,C 180,E1 24374.203,E2 24374.203} C_VEL
LIN {X 0,Y 248.781,Z 1226.068,A -85,B 0,C 180,E1 24383.003,E2 24383.003} C_VEL
LIN {X 0,Y 248.944,Z 1227.51,A -85,B 0,C 180,E1 24390,E2 24390} C_VEL
LIN {X 0,Y 248.78,Z 1226.081,A -85,B 0,C 180,E1 24396.997,E2 24396.997} C_VEL
LIN {X 0,Y 250.433,Z 1220.458,A -85,B 0,C 180,E1 24405.62,E2 24405.62} C_VEL
LIN {X 0,Y 255.961,Z 1208.747,A -85,B 0,C 180,E1 24415.416,E2 24415.416} C_VEL
LIN {X 0,Y 267.318,Z 1190.284,A -85,B 0,C 180,E1 24424.951,E2 24424.951} C_VEL
LIN {X 0,Y 282.836,Z 1166.378,A -85,B 0,C 180,E1 24433.084,E2 24433.084} C_VEL
LIN {X 0,Y 300.864,Z 1137.852,A -85,B 0,C 180,E1 24439.619,E2 24439.619} C_VEL
LIN {X 0,Y 319.894,Z 1104.304,A -85,B 0,C 180,E1 24444.867,E2 24444.867} C_VEL
LIN {X 0,Y 337.791,Z 1067.099,A -85,B 0,C 180,E1 24448.857,E2 24448.857} C_VEL
LIN {X 0,Y 351.69,Z 1030.228,A -85,B 0,C 180,E1 24451.714,E2 24451.714} C_VEL
LIN {X 0,Y 347.716,Z 1007.347,A -85,B 0,C 180,E1 24456.473,E2 24456.473} C_VEL
LIN {X 0,Y 342.27,Z 988.09,A -85,B 0,C 180,E1 24461.518,E2 24461.518} C_VEL
LIN {X 0,Y 336.575,Z 972.643,A -85,B 0,C 180,E1 24466.991,E2 24466.991} C_VEL
LIN {X 0,Y 332.163,Z 962.505,A -85,B 0,C 180,E1 24472.297,E2 24472.297} C_VEL
LIN {X 0,Y 330.391,Z 957.95,A -85,B 0,C 180,E1 24475.559,E2 24475.559} C_VEL
LIN {X 0,Y 329.169,Z 952.81,A -85,B 0,C 180,E1 24480.656,E2 24480.656} C_VEL
LIN {X 0,Y 329.191,Z 953.861,A -85,B 0,C 180,E1 24485.691,E2 24485.691} C_VEL
LIN {X 0,Y 332.067,Z 961.031,A -85,B 0,C 180,E1 24492.519,E2 24492.519} C_VEL
LIN {X 0,Y 336.688,Z 970.529,A -85,B 0,C 180,E1 24497.856,E2 24497.856} C_VEL
LIN {X 0,Y 342.074,Z 983.117,A -85,B 0,C 180,E1 24502.629,E2 24502.629} C_VEL
LIN {X 0,Y 343.481,Z 991.037,A -85,B 0,C 180,E1 24504.357,E2 24504.357} C_VEL
LIN {X 0,Y 344.514,Z 1006.454,A -85,B 0,C 180,E1 24507.018,E2 24507.018} C_VEL
LIN {X 0,Y 349.674,Z 1028.903,A -85,B 0,C 180,E1 24512.049,E2 24512.049} C_VEL
LIN {X 0,Y 349.312,Z 1033.446,A -85,B 0,C 180,E1 24512.651,E2 24512.651} C_VEL
LIN {X 0,Y 334.09,Z 1070.904,A -85,B 0,C 180,E1 24515.274,E2 24515.274} C_VEL
LIN {X 0,Y 316.514,Z 1105.072,A -85,B 0,C 180,E1 24518.82,E2 24518.82} C_VEL
LIN {X 0,Y 297.382,Z 1136.131,A -85,B 0,C 180,E1 24523.632,E2 24523.632} C_VEL
LIN {X 0,Y 278.676,Z 1162.57,A -85,B 0,C 180,E1 24529.782,E2 24529.782} C_VEL
LIN {X 0,Y 262.657,Z 1183.547,A -85,B 0,C 180,E1 24537.216,E2 24537.216} C_VEL
LIN {X 0,Y 250.636,Z 1199.246,A -85,B 0,C 180,E1 24545.916,E2 24545.916} C_VEL
LIN {X 0,Y 243.582,Z 1209.585,A -85,B 0,C 180,E1 24555.592,E2 24555.592} C_VEL
LIN {X 0,Y 241.347,Z 1213.671,A -85,B 0,C 180,E1 24562.787,E2 24562.787} C_VEL
LIN {X 0,Y 241.105,Z 1214.986,A -85,B 0,C 180,E1 24570,E2 24570} C_VEL
LIN {X 0,Y 241.372,Z 1213.606,A -85,B 0,C 180,E1 24577.213,E2 24577.213} C_VEL
LIN {X 0,Y 244.665,Z 1207.753,A -85,B 0,C 180,E1 24586.449,E2 24586.449} C_VEL
LIN {X 0,Y 252.85,Z 1196.091,A -85,B 0,C 180,E1 24596.024,E2 24596.024} C_VEL
LIN {X 0,Y 266.319,Z 1178.622,A -85,B 0,C 180,E1 24604.679,E2 24604.679} C_VEL
LIN {X 0,Y 282.668,Z 1156.82,A -85,B 0,C 180,E1 24611.654,E2 24611.654} C_VEL
LIN {X 0,Y 300.963,Z 1130.304,A -85,B 0,C 180,E1 24617.296,E2 24617.296} C_VEL
LIN {X 0,Y 319.312,Z 1099.591,A -85,B 0,C 180,E1 24621.726,E2 24621.726} C_VEL
LIN {X 0,Y 336.266,Z 1065.626,A -85,B 0,C 180,E1 24625.043,E2 24625.043} C_VEL
LIN {X 0,Y 349.89,Z 1030.805,A -85,B 0,C 180,E1 24627.44,E2 24627.44} C_VEL
LIN {X 0,Y 344.771,Z 1007.823,A -85,B 0,C 180,E1 24632.483,E2 24632.483} C_VEL
LIN {X 0,Y 338.837,Z 989.752,A -85,B 0,C 180,E1 24637.669,E2 24637.669} C_VEL
LIN {X 0,Y 332.967,Z 975.542,A -85,B 0,C 180,E1 24643.398,E2 24643.398} C_VEL
LIN {X 0,Y 328.634,Z 965.805,A -85,B 0,C 180,E1 24649.546,E2 24649.546} C_VEL
LIN {X 0,Y 327.206,Z 960.59,A -85,B 0,C 180,E1 24654.691,E2 24654.691} C_VEL
LIN {X 0,Y 327.224,Z 961.187,A -85,B 0,C 180,E1 24660.501,E2 24660.501} C_VEL
LIN {X 0,Y 329.366,Z 968.41,A -85,B 0,C 180,E1 24666.689,E2 24666.689} C_VEL
LIN {X 0,Y 333.134,Z 978.065,A -85,B 0,C 180,E1 24672.061,E2 24672.061} C_VEL
LIN {X 0,Y 338.231,Z 993.285,A -85,B 0,C 180,E1 24677.65,E2 24677.65} C_VEL
LIN {X 0,Y 343.379,Z 1013.22,A -85,B 0,C 180,E1 24683.054,E2 24683.054} C_VEL
LIN {X 0,Y 346.349,Z 1033.887,A -85,B 0,C 180,E1 24687.452,E2 24687.452} C_VEL
LIN {X 0,Y 330.832,Z 1072.317,A -85,B 0,C 180,E1 24690.496,E2 24690.496} C_VEL
LIN {X 0,Y 313.383,Z 1106.955,A -85,B 0,C 180,E1 24694.349,E2 24694.349} C_VEL
LIN {X 0,Y 294.521,Z 1139.016,A -85,B 0,C 180,E1 24699.489,E2 24699.489} C_VEL
LIN {X 0,Y 276.039,Z 1167.289,A -85,B 0,C 180,E1 24706.128,E2 24706.128} C_VEL
LIN {X 0,Y 260.092,Z 1190.799,A -85,B 0,C 180,E1 24714.366,E2 24714.366} C_VEL
LIN {X 0,Y 248.643,Z 1208.453,A -85,B 0,C 180,E1 24723.779,E2 24723.779} C_VEL
LIN {X 0,Y 242.72,Z 1220.041,A -85,B 0,C 180,E1 24733.684,E2 24733.684} C_VEL
LIN {X 0,Y 240.88,Z 1225.864,A -85,B 0,C 180,E1 24742.772,E2 24742.772} C_VEL
LIN {X 0,Y 241.053,Z 1227.308,A -85,B 0,C 180,E1 24750,E2 24750} C_VEL
LIN {X 0,Y 240.878,Z 1225.878,A -85,B 0,C 180,E1 24757.227,E2 24757.227} C_VEL
LIN {X 0,Y 242.739,Z 1220.085,A -85,B 0,C 180,E1 24766.314,E2 24766.314} C_VEL
LIN {X 0,Y 248.63,Z 1208.527,A -85,B 0,C 180,E1 24776.222,E2 24776.222} C_VEL
LIN {X 0,Y 260.76,Z 1189.901,A -85,B 0,C 180,E1 24786.041,E2 24786.041} C_VEL
LIN {X 0,Y 276.912,Z 1166.116,A -85,B 0,C 180,E1 24794.242,E2 24794.242} C_VEL
LIN {X 0,Y 295.645,Z 1137.554,A -85,B 0,C 180,E1 24800.824,E2 24800.824} C_VEL
LIN {X 0,Y 315.662,Z 1103.205,A -85,B 0,C 180,E1 24806.172,E2 24806.172} C_VEL
LIN {X 0,Y 334.151,Z 1065.571,A -85,B 0,C 180,E1 24810.141,E2 24810.141} C_VEL
LIN {X 0,Y 346.538,Z 1034.503,A -85,B 0,C 180,E1 24812.472,E2 24812.472} C_VEL
LIN {X 0,Y 343.451,Z 1012.922,A -85,B 0,C 180,E1 24817.074,E2 24817.074} C_VEL
LIN {X 0,Y 338.553,Z 993.734,A -85,B 0,C 180,E1 24822.267,E2 24822.267} C_VEL
LIN {X 0,Y 333.474,Z 978.787,A -85,B 0,C 180,E1 24827.785,E2 24827.785} C_VEL
LIN {X 0,Y 329.704,Z 969.025,A -85,B 0,C 180,E1 24833.152,E2 24833.152} C_VEL
LIN {X 0,Y 328.197,Z 965.218,A -85,B 0,C 180,E1 24836.192,E2 24836.192} C_VEL
LIN {X 0,Y 327.354,Z 960.479,A -85,B 0,C 180,E1 24841.322,E2 24841.322} C_VEL
LIN {X 0,Y 327.437,Z 961.656,A -85,B 0,C 180,E1 24845.638,E2 24845.638} C_VEL
LIN {X 0,Y 329.983,Z 968.428,A -85,B 0,C 180,E1 24852.219,E2 24852.219} C_VEL
LIN {X 0,Y 334.248,Z 978.092,A -85,B 0,C 180,E1 24857.644,E2 24857.644} C_VEL
LIN {X 0,Y 340.558,Z 994.176,A -85,B 0,C 180,E1 24863.596,E2 24863.596} C_VEL
LIN {X 0,Y 344.514,Z 1006.454,A -85,B 0,C 180,E1 24867.018,E2 24867.018} C_VEL
LIN {X 0,Y 345.138,Z 1015.509,A -85,B 0,C 180,E1 24868.594,E2 24868.594} C_VEL
LIN {X 0,Y 344.564,Z 1032.09,A -85,B 0,C 180,E1 24871.044,E2 24871.044} C_VEL
LIN {X 0,Y 344.217,Z 1036.496,A -85,B 0,C 180,E1 24871.689,E2 24871.689} C_VEL
LIN {X 0,Y 328.92,Z 1072.719,A -85,B 0,C 180,E1 24874.274,E2 24874.274} C_VEL
LIN {X 0,Y 311.12,Z 1106.212,A -85,B 0,C 180,E1 24877.791,E2 24877.791} C_VEL
LIN {X 0,Y 291.746,Z 1136.664,A -85,B 0,C 180,E1 24882.551,E2 24882.551} C_VEL
LIN {X 0,Y 272.624,Z 1162.813,A -85,B 0,C 180,E1 24888.701,E2 24888.701} C_VEL
LIN {X 0,Y 255.473,Z 1184.325,A -85,B 0,C 180,E1 24896.51,E2 24896.51} C_VEL
LIN {X 0,Y 243.346,Z 1199.458,A -85,B 0,C 180,E1 24905.146,E2 24905.146} C_VEL
LIN {X 0,Y 235.861,Z 1209.791,A -85,B 0,C 180,E1 24915.11,E2 24915.11} C_VEL
LIN {X 0,Y 233.476,Z 1213.874,A -85,B 0,C 180,E1 24922.542,E2 24922.542} C_VEL
LIN {X 0,Y 233.203,Z 1215.188,A -85,B 0,C 180,E1 24930,E2 24930} C_VEL
LIN {X 0,Y 233.504,Z 1213.81,A -85,B 0,C 180,E1 24937.458,E2 24937.458} C_VEL
LIN {X 0,Y 237.119,Z 1207.838,A -85,B 0,C 180,E1 24947.14,E2 24947.14} C_VEL
LIN {X 0,Y 245.679,Z 1196.302,A -85,B 0,C 180,E1 24956.844,E2 24956.844} C_VEL
LIN {X 0,Y 259.772,Z 1178.851,A -85,B 0,C 180,E1 24965.685,E2 24965.685} C_VEL
LIN {X 0,Y 276.174,Z 1157.85,A -85,B 0,C 180,E1 24972.542,E2 24972.542} C_VEL
LIN {X 0,Y 295.038,Z 1131.476,A -85,B 0,C 180,E1 24978.275,E2 24978.275} C_VEL
LIN {X 0,Y 314.128,Z 1100.563,A -85,B 0,C 180,E1 24982.79,E2 24982.79} C_VEL
LIN {X 0,Y 331.803,Z 1066.128,A -85,B 0,C 180,E1 24986.16,E2 24986.16} C_VEL
LIN {X 0,Y 344.631,Z 1034.782,A -85,B 0,C 180,E1 24988.302,E2 24988.302} C_VEL
LIN {X 0,Y 340.628,Z 1013.332,A -85,B 0,C 180,E1 24993.133,E2 24993.133} C_VEL
LIN {X 0,Y 334.854,Z 994.495,A -85,B 0,C 180,E1 24998.786,E2 24998.786} C_VEL
LIN {X 0,Y 329.358,Z 979.969,A -85,B 0,C 180,E1 25005.102,E2 25005.102} C_VEL
LIN {X 0,Y 326.39,Z 973.044,A -85,B 0,C 180,E1 25010.149,E2 25010.149} C_VEL
LIN {X 0,Y 325.369,Z 968.287,A -85,B 0,C 180,E1 25014.661,E2 25014.661} C_VEL
LIN {X 0,Y 325.335,Z 968.823,A -85,B 0,C 180,E1 25020.337,E2 25020.337} C_VEL
LIN {X 0,Y 327.069,Z 976.021,A -85,B 0,C 180,E1 25026.57,E2 25026.57} C_VEL
LIN {X 0,Y 330.512,Z 985.647,A -85,B 0,C 180,E1 25031.907,E2 25031.907} C_VEL
LIN {X 0,Y 335.266,Z 1001.752,A -85,B 0,C 180,E1 25037.811,E2 25037.811} C_VEL
LIN {X 0,Y 339.526,Z 1021.7,A -85,B 0,C 180,E1 25043.162,E2 25043.162} C_VEL
LIN {X 0,Y 341.321,Z 1037.252,A -85,B 0,C 180,E1 25046.53,E2 25046.53} C_VEL
LIN {X 0,Y 323.817,Z 1078.159,A -85,B 0,C 180,E1 25049.855,E2 25049.855} C_VEL
LIN {X 0,Y 303.93,Z 1115.397,A -85,B 0,C 180,E1 25054.335,E2 25054.335} C_VEL
LIN {X 0,Y 282.831,Z 1148.716,A -85,B 0,C 180,E1 25060.31,E2 25060.31} C_VEL
LIN {X 0,Y 264.546,Z 1175.04,A -85,B 0,C 180,E1 25067.398,E2 25067.398} C_VEL
LIN {X 0,Y 248.34,Z 1197.748,A -85,B 0,C 180,E1 25076.691,E2 25076.691} C_VEL
LIN {X 0,Y 238.139,Z 1213.588,A -85,B 0,C 180,E1 25086.941,E2 25086.941} C_VEL
LIN {X 0,Y 234.095,Z 1222.143,A -85,B 0,C 180,E1 25096.115,E2 25096.115} C_VEL
LIN {X 0,Y 232.894,Z 1226.738,A -85,B 0,C 180,E1 25106.269,E2 25106.269} C_VEL
LIN {X 0,Y 233.147,Z 1227.106,A -85,B 0,C 180,E1 25110,E2 25110} C_VEL
LIN {X 0,Y 232.981,Z 1225.675,A -85,B 0,C 180,E1 25117.474,E2 25117.474} C_VEL
LIN {X 0,Y 235.007,Z 1219.875,A -85,B 0,C 180,E1 25126.867,E2 25126.867} C_VEL
LIN {X 0,Y 241.315,Z 1208.387,A -85,B 0,C 180,E1 25137.024,E2 25137.024} C_VEL
LIN {X 0,Y 253.51,Z 1190.668,A -85,B 0,C 180,E1 25146.707,E2 25146.707} C_VEL
LIN {X 0,Y 270.922,Z 1166.154,A -85,B 0,C 180,E1 25155.363,E2 25155.363} C_VEL
LIN {X 0,Y 290.568,Z 1137.252,A -85,B 0,C 180,E1 25162.069,E2 25162.069} C_VEL
LIN {X 0,Y 311.367,Z 1102.514,A -85,B 0,C 180,E1 25167.455,E2 25167.455} C_VEL
LIN {X 0,Y 330.061,Z 1065.37,A -85,B 0,C 180,E1 25171.333,E2 25171.333} C_VEL
LIN {X 0,Y 341.554,Z 1037.224,A -85,B 0,C 180,E1 25173.49,E2 25173.49} C_VEL
LIN {X 0,Y 338.45,Z 1014.838,A -85,B 0,C 180,E1 25178.574,E2 25178.574} C_VEL
LIN {X 0,Y 333.843,Z 995.848,A -85,B 0,C 180,E1 25184.197,E2 25184.197} C_VEL
LIN {X 0,Y 329.701,Z 982.88,A -85,B 0,C 180,E1 25189.573,E2 25189.573} C_VEL
LIN {X 0,Y 326.433,Z 973.235,A -85,B 0,C 180,E1 25195.671,E2 25195.671} C_VEL
LIN {X 0,Y 325.514,Z 968.142,A -85,B 0,C 180,E1 25201.33,E2 25201.33} C_VEL
LIN {X 0,Y 325.552,Z 969.352,A -85,B 0,C 180,E1 25205.504,E2 25205.504} C_VEL
LIN {X 0,Y 327.826,Z 976.083,A -85,B 0,C 180,E1 25212.095,E2 25212.095} C_VEL
LIN {X 0,Y 331.65,Z 985.458,A -85,B 0,C 180,E1 25217.378,E2 25217.378} C_VEL
LIN {X 0,Y 337.52,Z 1001.825,A -85,B 0,C 180,E1 25223.47,E2 25223.47} C_VEL
LIN {X 0,Y 342.57,Z 1021.309,A -85,B 0,C 180,E1 25228.661,E2 25228.661} C_VEL
LIN {X 0,Y 344.564,Z 1032.09,A -85,B 0,C 180,E1 25231.044,E2 25231.044} C_VEL
LIN {X 0,Y 342.817,Z 1038.051,A -85,B 0,C 180,E1 25231.525,E2 25231.525} C_VEL
LIN {X 0,Y 333.764,Z 1052.968,A -85,B 0,C 180,E1 25231.555,E2 25231.555} C_VEL
LIN {X 0,Y 316.384,Z 1088.898,A -85,B 0,C 180,E1 25234.596,E2 25234.596} C_VEL
LIN {X 0,Y 297.786,Z 1120.164,A -85,B 0,C 180,E1 25238.523,E2 25238.523} C_VEL
LIN {X 0,Y 278.046,Z 1148.343,A -85,B 0,C 180,E1 25243.773,E2 25243.773} C_VEL
LIN {X 0,Y 259.111,Z 1172.2,A -85,B 0,C 180,E1 25250.508,E2 25250.508} C_VEL
LIN {X 0,Y 244.281,Z 1189.937,A -85,B 0,C 180,E1 25258.18,E2 25258.18} C_VEL
LIN {X 0,Y 232.573,Z 1204.099,A -85,B 0,C 180,E1 25267.999,E2 25267.999} C_VEL
LIN {X 0,Y 226.581,Z 1212.388,A -85,B 0,C 180,E1 25278.427,E2 25278.427} C_VEL
LIN {X 0,Y 225.231,Z 1215.075,A -85,B 0,C 180,E1 25286.143,E2 25286.143} C_VEL
LIN {X 0,Y 225.245,Z 1215.041,A -85,B 0,C 180,E1 25293.858,E2 25293.858} C_VEL
LIN {X 0,Y 227.376,Z 1211.138,A -85,B 0,C 180,E1 25303.489,E2 25303.489} C_VEL
LIN {X 0,Y 234.317,Z 1201.741,A -85,B 0,C 180,E1 25313.84,E2 25313.84} C_VEL
LIN {X 0,Y 247.182,Z 1186.342,A -85,B 0,C 180,E1 25323.486,E2 25323.486} C_VEL
LIN {X 0,Y 263.52,Z 1166.73,A -85,B 0,C 180,E1 25331.161,E2 25331.161} C_VEL
LIN {X 0,Y 282.624,Z 1141.932,A -85,B 0,C 180,E1 25337.495,E2 25337.495} C_VEL
LIN {X 0,Y 302.286,Z 1112.798,A -85,B 0,C 180,E1 25342.434,E2 25342.434} C_VEL
LIN {X 0,Y 321.299,Z 1079.249,A -85,B 0,C 180,E1 25346.225,E2 25346.225} C_VEL
LIN {X 0,Y 338.004,Z 1042.184,A -85,B 0,C 180,E1 25349.035,E2 25349.035} C_VEL
LIN {X 0,Y 339.511,Z 1038.231,A -85,B 0,C 180,E1 25349.262,E2 25349.262} C_VEL
LIN {X 0,Y 336.31,Z 1018.206,A -85,B 0,C 180,E1 25353.952,E2 25353.952} C_VEL
LIN {X 0,Y 331.577,Z 1001.101,A -85,B 0,C 180,E1 25359.267,E2 25359.267} C_VEL
LIN {X 0,Y 327.1,Z 988.285,A -85,B 0,C 180,E1 25364.914,E2 25364.914} C_VEL
LIN {X 0,Y 324.113,Z 980.54,A -85,B 0,C 180,E1 25370.291,E2 25370.291} C_VEL
LIN {X 0,Y 323.123,Z 975.824,A -85,B 0,C 180,E1 25375.637,E2 25375.637} C_VEL
LIN {X 0,Y 323.163,Z 976.607,A -85,B 0,C 180,E1 25380.339,E2 25380.339} C_VEL
LIN {X 0,Y 324.623,Z 983.244,A -85,B 0,C 180,E1 25386.199,E2 25386.199} C_VEL
LIN {X 0,Y 327.84,Z 993.693,A -85,B 0,C 180,E1 25392.005,E2 25392.005} C_VEL
LIN {X 0,Y 332.096,Z 1010.278,A -85,B 0,C 180,E1 25397.987,E2 25397.987} C_VEL
LIN {X 0,Y 335.22,Z 1028.809,A -85,B 0,C 180,E1 25402.944,E2 25402.944} C_VEL
